Universal Robots PolyScope program: DAS428_958_02_MAR_21_DAS_lado_derecho_jig2.urp

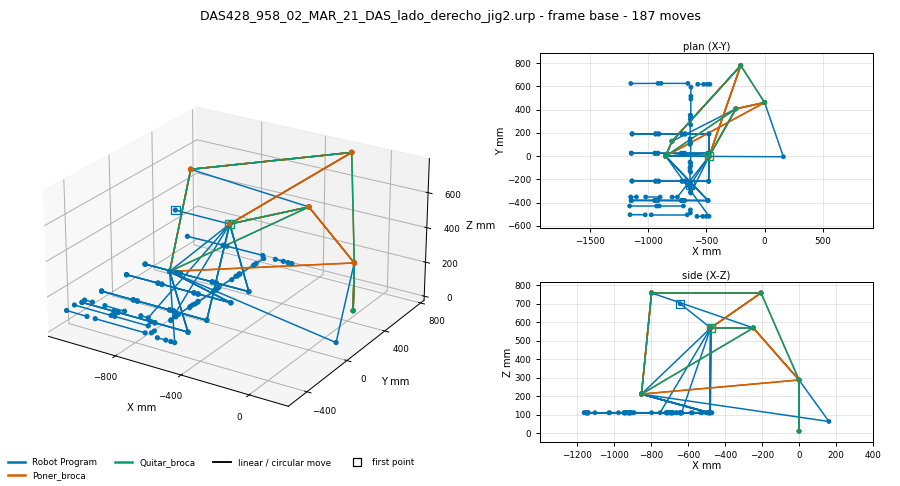
[picture p0: tool path of DAS428_958_02_MAR_21_DAS_lado_derecho_jig2.urp in frame base, 187 of 372 moves have a stored position in this frame; points joined in program order, loops and branches not executed]
Program DAS428_958_02_MAR_21_DAS_lado_derecho_jig2 (installation=instalacion_26_FEB_21 directory=/programs/jig2/derecha createdIn=5.6.0.90886 lastSavedIn=5.6.0.90886 robotSerialNumber=20195001785)
Calibrated DH parameters: a=[0.000107, -0.568984, -0.552934, -0.00001, -0.000063, 0]; d=[0.180718, -257.998067, 200.685024, 57.48776, 0.119923, 0.115353]; alpha=[1.571119, 0.000876, -0.002498, 1.571178, -1.570523, 0]; deltaTheta=[0, -0.378191, 0.631587, -0.253396, 0, 0]
Robot Program (runOnlyOnce=false)
  Folder Variables
    bajada_broca := p[0,0,-0.008,0,0,0]
    barrenos_menos1 := 0
    barreno_actual := 0
    posicion := p[0,0,300,0,0,0]
    cambiar_broca := False
    barrenos_hechos := 0
    eje7 := 0
    Wait Sleep waitTime=0.5
  Folder Home
    Wait Sleep waitTime=0.3
    MoveL speed 250 mm/s, acceleration 1200 mm/s^2 (useActiveTCP=true) feature=Base
      Waypoint Traslacion: TCP in base x=-641.047 y=-250.866 z=699.551 mm, rx=2.5572 ry=-1.7056 rz=-0.147 rad; joints [-0.465, -94.502, 70.676, 17.843, -302.102, -0.163] deg; TCP offset x=0.411 y=-218.298 z=37.994 mm, rx=1.558 ry=-0.1255 rz=0.1212 rad
      Waypoint Home2: TCP in base x=-476.229 y=0 z=568.737 mm, rx=2.0263 ry=-2.3929 rz=-0.0208 rad; joints [-32.551, -116.469, 98.413, 17.843, -302.102, -0.163] deg; TCP offset x=0.411 y=-218.298 z=37.994 mm, rx=1.558 ry=-0.1255 rz=0.1212 rad
      Waypoint Home3: TCP in base x=-850.182 y=0 z=211.32 mm, rx=-2.0297 ry=2.3968 rz=0.0066 rad; joints [-14.374, -75.698, 98.757, -22.649, -284.037, -0.192] deg; TCP offset x=0.411 y=-218.298 z=37.994 mm, rx=1.558 ry=-0.1255 rz=0.1212 rad
      Waypoint Home4: TCP in base x=-850.182 y=0 z=211.32 mm, rx=-2.0297 ry=2.3968 rz=0.0066 rad; joints [-14.374, -75.698, 98.757, -22.649, -284.037, -0.192] deg; TCP offset x=0.411 y=-218.298 z=37.994 mm, rx=1.558 ry=-0.1255 rz=0.1212 rad
      Waypoint PosicionApagado: TCP in base x=162.343 y=-4.969 z=63.23 mm, rx=-1.8392 ry=0.2253 rz=0.1717 rad; joints [89.997, -89.982, 149.522, 14.976, -265, 0.001] deg
      Waypoint Precambio_broca: TCP in base x=0.83 y=461.518 z=287.521 mm, rx=-0.2218 ry=-3.132 rz=0.0004 rad; joints [-125.124, -120.118, 128.54, -7.699, -306.118, -0.232] deg; TCP offset x=0.411 y=-218.298 z=37.994 mm, rx=1.558 ry=-0.1255 rz=0.1212 rad
      Waypoint yendo1: TCP in base x=-246.137 y=407.69 z=568.737 mm, rx=-0.5894 ry=3.0844 rz=0.0228 rad; joints [-91.431, -116.469, 98.413, 17.843, -302.102, -0.163] deg
      Waypoint Precam_bro1: TCP in base x=-795.771 y=128.511 z=757.632 mm, rx=1.5534 ry=-2.1987 rz=-0.8089 rad; joints [-24.356, -99.239, 84.164, -22.649, -284.037, -0.192] deg; TCP offset x=0.411 y=-218.298 z=37.994 mm, rx=1.558 ry=-0.1255 rz=0.1212 rad
      Waypoint Precam_bro2: TCP in base x=-204.472 y=779.716 z=757.632 mm, rx=-0.1114 ry=2.934 rz=1.0184 rad; joints [-90.488, -99.239, 84.164, -22.649, -284.037, -0.192] deg
    SafeHome (positionOptionType=SPEED_AND_ACCELERATION speed=1.047198 acceleration=1.396263 nextMotionTime=2)
    SuppressedNode
      If eje7≟3
        MoveL speed 250 mm/s, acceleration 1200 mm/s^2 (useActiveTCP=true) feature=Base
          MoveDirectionNode (selectedDirection=ZPlus)
            Until DISTANCE (allowActions=false deceleration=3 distanceNodeType=STOP) Distance=0.1; motionParameters(blendRadius=0)
          Waypoint Home3: TCP in base x=-850.182 y=0 z=211.32 mm, rx=-2.0297 ry=2.3968 rz=0.0066 rad; joints [-14.374, -75.698, 98.757, -22.649, -284.037, -0.192] deg
    SuppressedNode
      MoveL speed 250 mm/s, acceleration 1200 mm/s^2 (useActiveTCP=true) feature=Base
        Waypoint home_trans: TCP in base x=-171.077 y=546.65 z=109.574 mm, rx=0.1544 ry=3.1247 rz=-0.2011 rad; joints [-91.802, -93.053, 127.954, -27.005, -275.278, -0.192] deg; TCP offset x=0.411 y=-218.298 z=37.994 mm, rx=1.558 ry=-0.1255 rz=0.1212 rad
    Wait Sleep waitTime=0.3
    iniciando_prog := True
    Call Poner_broca
  Folder Posicion2
    Folder Inicio
      eje7 := 2
      MoveL speed 250 mm/s, acceleration 1200 mm/s^2 (useActiveTCP=true) feature=Base
        Waypoint Home2: TCP in base x=-476.229 y=0 z=568.737 mm, rx=2.0263 ry=-2.3929 rz=-0.0208 rad; joints [-32.551, -116.469, 98.413, 17.843, -302.102, -0.163] deg
    Folder SeatTracks
      Folder Broca_1
        Folder Linea1
          Folder Marcar_puntos
            MoveL speed 100 mm/s, acceleration 500 mm/s^2 (useActiveTCP=true) feature=Base
              Waypoint Home2: TCP in base x=-476.229 y=0 z=568.737 mm, rx=2.0263 ry=-2.3929 rz=-0.0208 rad; joints [-32.551, -116.469, 98.413, 17.843, -302.102, -0.163] deg
              SuppressedNode
                Folder var
                  barrenos_hechos := 10
                  eje7 := 2
                  cambiar_broca := False
                  iniciando_prog := False
              SuppressedNode
                iniciando_prog := False
              SuppressedNode
                Call Poner_broca
              Waypoint Linea1_A: TCP in base x=-480.065 y=-215.567 z=110.155 mm, rx=2.0263 ry=-2.3929 rz=-0.0208 rad; joints [7.208, -100.641, 136.552, -36.178, -262.472, -0.269] deg; TCP offset x=0.411 y=-218.298 z=37.994 mm, rx=1.558 ry=-0.1255 rz=0.1212 rad
              Waypoint Linea1_B: TCP in base x=-683.26 y=-215.006 z=110.473 mm, rx=2.0263 ry=-2.3929 rz=-0.0208 rad; joints [4.504, -82.11, 118.563, -36.711, -265.183, -0.242] deg
              Waypoint Linea1_C: TCP in base x=-708.66 y=-214.986 z=110.511 mm, rx=2.0264 ry=-2.3929 rz=-0.0208 rad; joints [4.302, -80.013, 116.028, -36.271, -265.387, -0.241] deg
              Waypoint Linea1_D: TCP in base x=-911.542 y=-214.533 z=110.306 mm, rx=2.0263 ry=-2.3929 rz=-0.0209 rad; joints [3.146, -63.772, 93.392, -29.877, -266.531, -0.235] deg
              Waypoint Linea1_E: TCP in base x=-936.518 y=-214.589 z=110.515 mm, rx=2.0263 ry=-2.3929 rz=-0.0209 rad; joints [3.051, -61.764, 90.233, -28.728, -266.622, -0.234] deg
              Waypoint Linea1_F: TCP in base x=-1139.514 y=-213.881 z=110.127 mm, rx=2.0263 ry=-2.3929 rz=-0.0209 rad; joints [2.389, -43.641, 59.472, -16.09, -267.256, -0.236] deg
          Folder AB
            'desbaste_inicial'
            bajada_broca := p[0,0,-0.008,0,0,0]
            barrenos_menos1 := 8
            barreno_actual := 0
            Loop While (checkContinuously=false) expression=barreno_actual≤barrenos_menos1
              Folder Perforacion
                MoveL speed 100 mm/s, acceleration 500 mm/s^2 (useActiveTCP=true) feature=Base
                  internos := interpolate_pose(Linea1_A, Linea1_B, barreno_actual/barrenos_menos1)
                  Waypoint Waypoint (Variable): variable=internos
                  'desbaste_inicial'
                  bajada_broca := p[0,0,-0.008,0,0,0]
                  bajada := p[0,0,0.008,0,0,0]
                  MoveDirectionNode (selectedDirection=ZMinus toolParams=0.03, 0.035)
                    Until DISTANCE (allowActions=false deceleration=3 distanceNodeType=STOP) Distance=0.076; motionParameters(blendRadius=0)
                  Popup Message (haltProgram=false message=punto contacto alanzdo inputType=Text)
                  MoveDirectionNode (selectedDirection=ZPlus toolParams=0.003, 0.005)
                    Until DISTANCE (allowActions=false deceleration=3 distanceNodeType=STOP) Distance=0.002; motionParameters(blendRadius=0)
                  Wait Sleep waitTime=0.3
                  Set DigitalOutput pin=config_out[1]; digitalValue=1
                  Wait Sleep waitTime=0.3
                  Loop Counting (count=3) loopVariable(name=Loop_39)
                    bajar := pose_add(get_actual_tcp_pose(), bajada_broca)
                    Waypoint Waypoint (Variable): motionParameters(jointSpeed=1.047198 jointAcceleration=1.396263 cartesianSpeed=0.001 cartesianAcceleration=0.005); variable=bajar
                    subir := pose_sub(get_actual_tcp_pose(), bajada_broca)
                    Waypoint Waypoint (Variable): motionParameters(jointSpeed=1.047198 jointAcceleration=1.396263 cartesianSpeed=0.005 cartesianAcceleration=0.01); variable=subir
                    bajada_broca := pose_sub(bajada_broca, bajada)
                  MoveDirectionNode (selectedDirection=ZPlus toolParams=0.03, 0.035)
                    Until DISTANCE (allowActions=false deceleration=3 distanceNodeType=STOP) Distance=0.06; motionParameters(blendRadius=0)
                  Set DigitalOutput pin=config_out[1]; digitalValue=0
                  barreno_actual := barreno_actual+1
                  Call Quitar_broca
                  Call Poner_broca
          Folder CD
            'desbaste_inicial'
            bajada_broca := p[0,0,-0.008,0,0,0]
            barrenos_menos1 := 8
            barreno_actual := 0
            Loop While (checkContinuously=false) expression=barreno_actual≤barrenos_menos1
              Folder Perforacion
                MoveL speed 100 mm/s, acceleration 500 mm/s^2 (useActiveTCP=true) feature=Base
                  internos := interpolate_pose(Linea1_C, Linea1_D, barreno_actual/barrenos_menos1)
                  Waypoint Waypoint (Variable): variable=internos
                  'desbaste_inicial'
                  bajada_broca := p[0,0,-0.008,0,0,0]
                  bajada := p[0,0,0.008,0,0,0]
                  MoveDirectionNode (selectedDirection=ZMinus toolParams=0.03, 0.035)
                    Until DISTANCE (allowActions=false deceleration=3 distanceNodeType=STOP) Distance=0.076; motionParameters(blendRadius=0)
                  Popup Message (haltProgram=false message=punto contacto alanzdo inputType=Text)
                  MoveDirectionNode (selectedDirection=ZPlus toolParams=0.003, 0.005)
                    Until DISTANCE (allowActions=false deceleration=3 distanceNodeType=STOP) Distance=0.002; motionParameters(blendRadius=0)
                  Wait Sleep waitTime=0.3
                  Set DigitalOutput pin=config_out[1]; digitalValue=1
                  Wait Sleep waitTime=0.3
                  Loop Counting (count=3) loopVariable(name=Loop_56)
                    bajar := pose_add(get_actual_tcp_pose(), bajada_broca)
                    Waypoint Waypoint (Variable): motionParameters(jointSpeed=1.047198 jointAcceleration=1.396263 cartesianSpeed=0.001 cartesianAcceleration=0.005); variable=bajar
                    subir := pose_sub(get_actual_tcp_pose(), bajada_broca)
                    Waypoint Waypoint (Variable): motionParameters(jointSpeed=1.047198 jointAcceleration=1.396263 cartesianSpeed=0.005 cartesianAcceleration=0.01); variable=subir
                    bajada_broca := pose_sub(bajada_broca, bajada)
                  MoveDirectionNode (selectedDirection=ZPlus toolParams=0.03, 0.035)
                    Until DISTANCE (allowActions=false deceleration=3 distanceNodeType=STOP) Distance=0.06; motionParameters(blendRadius=0)
                  Set DigitalOutput pin=config_out[1]; digitalValue=0
                  barreno_actual := barreno_actual+1
                  Call Quitar_broca
                  Call Poner_broca
          Folder EF
            'desbaste_inicial'
            bajada_broca := p[0,0,-0.008,0,0,0]
            barrenos_menos1 := 8
            barreno_actual := 0
            Loop While (checkContinuously=false) expression=barreno_actual≤barrenos_menos1
              Folder Perforacion
                MoveL speed 100 mm/s, acceleration 500 mm/s^2 (useActiveTCP=true) feature=Base
                  internos := interpolate_pose(Linea1_E, Linea1_F, barreno_actual/barrenos_menos1)
                  Waypoint Waypoint (Variable): variable=internos
                  'desbaste_inicial'
                  bajada_broca := p[0,0,-0.008,0,0,0]
                  bajada := p[0,0,0.008,0,0,0]
                  MoveDirectionNode (selectedDirection=ZMinus toolParams=0.03, 0.035)
                    Until DISTANCE (allowActions=false deceleration=3 distanceNodeType=STOP) Distance=0.067; motionParameters(blendRadius=0)
                  Popup Message (haltProgram=false message=punto contacto alanzdo inputType=Text)
                  MoveDirectionNode (selectedDirection=ZPlus toolParams=0.003, 0.005)
                    Until DISTANCE (allowActions=false deceleration=3 distanceNodeType=STOP) Distance=0.002; motionParameters(blendRadius=0)
                  Wait Sleep waitTime=0.3
                  Set DigitalOutput pin=config_out[1]; digitalValue=1
                  Wait Sleep waitTime=0.3
                  Loop Counting (count=3) loopVariable(name=Loop_61)
                    bajar := pose_add(get_actual_tcp_pose(), bajada_broca)
                    Waypoint Waypoint (Variable): motionParameters(jointSpeed=1.047198 jointAcceleration=1.396263 cartesianSpeed=0.001 cartesianAcceleration=0.005); variable=bajar
                    subir := pose_sub(get_actual_tcp_pose(), bajada_broca)
                    Waypoint Waypoint (Variable): motionParameters(jointSpeed=1.047198 jointAcceleration=1.396263 cartesianSpeed=0.005 cartesianAcceleration=0.01); variable=subir
                    bajada_broca := pose_sub(bajada_broca, bajada)
                  MoveDirectionNode (selectedDirection=ZPlus toolParams=0.03, 0.035)
                    Until DISTANCE (allowActions=false deceleration=3 distanceNodeType=STOP) Distance=0.06; motionParameters(blendRadius=0)
                  Set DigitalOutput pin=config_out[1]; digitalValue=0
                  barreno_actual := barreno_actual+1
                  Call Quitar_broca
                  Call Poner_broca
        Popup Message (haltProgram=false message=Linea1 con chica Terminada! inputType=Text)
        Folder Linea2
          Folder Marcar_puntos
            MoveL speed 100 mm/s, acceleration 500 mm/s^2 (useActiveTCP=true) feature=Base
              Waypoint Home2: TCP in base x=-476.229 y=0 z=568.737 mm, rx=2.0263 ry=-2.3929 rz=-0.0208 rad; joints [-32.551, -116.469, 98.413, 17.843, -302.102, -0.163] deg; TCP offset x=0.411 y=-218.298 z=37.994 mm, rx=1.558 ry=-0.1255 rz=0.1212 rad
              Waypoint Linea2_A: TCP in base x=-478.57 y=191.006 z=110.523 mm, rx=2.0263 ry=-2.3928 rz=-0.0209 rad; joints [-57.982, -102.694, 138.014, -35.673, -327.66, 0.098] deg; TCP offset x=0.411 y=-218.298 z=37.994 mm, rx=1.558 ry=-0.1255 rz=0.1212 rad
              Waypoint Linea2_B: TCP in base x=-681.936 y=191.002 z=110.452 mm, rx=2.0263 ry=-2.3929 rz=-0.0209 rad; joints [-37.869, -83.103, 119.731, -36.904, -307.554, -0.038] deg
              Waypoint Linea2_C: TCP in base x=-707.214 y=190.995 z=110.603 mm, rx=2.0262 ry=-2.3929 rz=-0.0208 rad; joints [-36.266, -80.967, 117.182, -36.489, -305.951, -0.043] deg
              Waypoint Linea2_D: TCP in base x=-910.192 y=191.479 z=110.348 mm, rx=2.0262 ry=-2.3928 rz=-0.0209 rad; joints [-27.02, -64.45, 94.432, -30.243, -296.696, -0.089] deg
              Waypoint Linea2_E: TCP in base x=-935.62 y=191.519 z=110.454 mm, rx=2.0261 ry=-2.3928 rz=-0.021 rad; joints [-26.177, -62.39, 91.226, -29.103, -295.849, -0.094] deg
              Waypoint Linea2_F: TCP in base x=-1138.395 y=191.499 z=110.212 mm, rx=2.0262 ry=-2.3928 rz=-0.021 rad; joints [-20.933, -44.304, 60.66, -16.618, -290.578, -0.121] deg
          Folder AB
            'desbaste_inicial'
            bajada_broca := p[0,0,-0.008,0,0,0]
            barrenos_menos1 := 8
            barreno_actual := 0
            Loop While (checkContinuously=false) expression=barreno_actual≤barrenos_menos1
              Folder Perforacion
                MoveL speed 100 mm/s, acceleration 500 mm/s^2 (useActiveTCP=true) feature=Base
                  internos := interpolate_pose(Linea2_A, Linea2_B, barreno_actual/barrenos_menos1)
                  Waypoint Waypoint (Variable): variable=internos
                  'desbaste_inicial'
                  bajada_broca := p[0,0,-0.008,0,0,0]
                  bajada := p[0,0,0.008,0,0,0]
                  MoveDirectionNode (selectedDirection=ZMinus toolParams=0.03, 0.035)
                    Until DISTANCE (allowActions=false deceleration=3 distanceNodeType=STOP) Distance=0.076; motionParameters(blendRadius=0)
                  Popup Message (haltProgram=false message=punto contacto alanzdo inputType=Text)
                  MoveDirectionNode (selectedDirection=ZPlus toolParams=0.003, 0.005)
                    Until DISTANCE (allowActions=false deceleration=3 distanceNodeType=STOP) Distance=0.002; motionParameters(blendRadius=0)
                  Wait Sleep waitTime=0.3
                  Set DigitalOutput pin=config_out[1]; digitalValue=1
                  Wait Sleep waitTime=0.3
                  Loop Counting (count=3) loopVariable(name=Loop_63)
                    bajar := pose_add(get_actual_tcp_pose(), bajada_broca)
                    Waypoint Waypoint (Variable): motionParameters(jointSpeed=1.047198 jointAcceleration=1.396263 cartesianSpeed=0.001 cartesianAcceleration=0.005); variable=bajar
                    subir := pose_sub(get_actual_tcp_pose(), bajada_broca)
                    Waypoint Waypoint (Variable): motionParameters(jointSpeed=1.047198 jointAcceleration=1.396263 cartesianSpeed=0.005 cartesianAcceleration=0.01); variable=subir
                    bajada_broca := pose_sub(bajada_broca, bajada)
                  MoveDirectionNode (selectedDirection=ZPlus toolParams=0.03, 0.035)
                    Until DISTANCE (allowActions=false deceleration=3 distanceNodeType=STOP) Distance=0.06; motionParameters(blendRadius=0)
                  Set DigitalOutput pin=config_out[1]; digitalValue=0
                  barreno_actual := barreno_actual+1
                  Call Quitar_broca
                  Call Poner_broca
          Folder CD
            'desbaste_inicial'
            bajada_broca := p[0,0,-0.008,0,0,0]
            barrenos_menos1 := 8
            barreno_actual := 0
            Loop While (checkContinuously=false) expression=barreno_actual≤barrenos_menos1
              Folder Perforacion
                MoveL speed 100 mm/s, acceleration 500 mm/s^2 (useActiveTCP=true) feature=Base
                  internos := interpolate_pose(Linea2_C, Linea2_D, barreno_actual/barrenos_menos1)
                  Waypoint Waypoint (Variable): variable=internos
                  'desbaste_inicial'
                  bajada_broca := p[0,0,-0.008,0,0,0]
                  bajada := p[0,0,0.008,0,0,0]
                  MoveDirectionNode (selectedDirection=ZMinus toolParams=0.03, 0.035)
                    Until DISTANCE (allowActions=false deceleration=3 distanceNodeType=STOP) Distance=0.076; motionParameters(blendRadius=0)
                  Popup Message (haltProgram=false message=punto contacto alanzdo inputType=Text)
                  MoveDirectionNode (selectedDirection=ZPlus toolParams=0.003, 0.005)
                    Until DISTANCE (allowActions=false deceleration=3 distanceNodeType=STOP) Distance=0.002; motionParameters(blendRadius=0)
                  Wait Sleep waitTime=0.3
                  Set DigitalOutput pin=config_out[1]; digitalValue=1
                  Wait Sleep waitTime=0.3
                  Loop Counting (count=3) loopVariable(name=Loop_65)
                    bajar := pose_add(get_actual_tcp_pose(), bajada_broca)
                    Waypoint Waypoint (Variable): motionParameters(jointSpeed=1.047198 jointAcceleration=1.396263 cartesianSpeed=0.001 cartesianAcceleration=0.005); variable=bajar
                    subir := pose_sub(get_actual_tcp_pose(), bajada_broca)
                    Waypoint Waypoint (Variable): motionParameters(jointSpeed=1.047198 jointAcceleration=1.396263 cartesianSpeed=0.005 cartesianAcceleration=0.01); variable=subir
                    bajada_broca := pose_sub(bajada_broca, bajada)
                  MoveDirectionNode (selectedDirection=ZPlus toolParams=0.03, 0.035)
                    Until DISTANCE (allowActions=false deceleration=3 distanceNodeType=STOP) Distance=0.06; motionParameters(blendRadius=0)
                  Set DigitalOutput pin=config_out[1]; digitalValue=0
                  barreno_actual := barreno_actual+1
                  Call Quitar_broca
                  Call Poner_broca
          Folder EF
            'desbaste_inicial'
            bajada_broca := p[0,0,-0.008,0,0,0]
            barrenos_menos1 := 8
            barreno_actual := 0
            Loop While (checkContinuously=false) expression=barreno_actual≤barrenos_menos1
              Folder Perforacion
                MoveL speed 100 mm/s, acceleration 500 mm/s^2 (useActiveTCP=true) feature=Base
                  internos := interpolate_pose(Linea2_E, Linea2_F, barreno_actual/barrenos_menos1)
                  Waypoint Waypoint (Variable): variable=internos
                  'desbaste_inicial'
                  bajada_broca := p[0,0,-0.008,0,0,0]
                  bajada := p[0,0,0.008,0,0,0]
                  MoveDirectionNode (selectedDirection=ZMinus toolParams=0.03, 0.035)
                    Until DISTANCE (allowActions=false deceleration=3 distanceNodeType=STOP) Distance=0.076; motionParameters(blendRadius=0)
                  Popup Message (haltProgram=false message=punto contacto alanzdo inputType=Text)
                  MoveDirectionNode (selectedDirection=ZPlus toolParams=0.003, 0.005)
                    Until DISTANCE (allowActions=false deceleration=3 distanceNodeType=STOP) Distance=0.002; motionParameters(blendRadius=0)
                  Wait Sleep waitTime=0.3
                  Set DigitalOutput pin=config_out[1]; digitalValue=1
                  Wait Sleep waitTime=0.3
                  Loop Counting (count=3) loopVariable(name=Loop_67)
                    bajar := pose_add(get_actual_tcp_pose(), bajada_broca)
                    Waypoint Waypoint (Variable): motionParameters(jointSpeed=1.047198 jointAcceleration=1.396263 cartesianSpeed=0.001 cartesianAcceleration=0.005); variable=bajar
                    subir := pose_sub(get_actual_tcp_pose(), bajada_broca)
                    Waypoint Waypoint (Variable): motionParameters(jointSpeed=1.047198 jointAcceleration=1.396263 cartesianSpeed=0.005 cartesianAcceleration=0.01); variable=subir
                    bajada_broca := pose_sub(bajada_broca, bajada)
                  MoveDirectionNode (selectedDirection=ZPlus toolParams=0.03, 0.035)
                    Until DISTANCE (allowActions=false deceleration=3 distanceNodeType=STOP) Distance=0.06; motionParameters(blendRadius=0)
                  Set DigitalOutput pin=config_out[1]; digitalValue=0
                  barreno_actual := barreno_actual+1
                  If barreno_actual>barrenos_menos1
                    cambiar_broca := True
                  Call Quitar_broca
                  Call Poner_broca
        Popup Message (haltProgram=false message=Linea2 con chica Terminada! inputType=Text)
      Folder Broca_2
        Folder Linea1
          Folder Marcar_puntos
            MoveL speed 100 mm/s, acceleration 500 mm/s^2 (useActiveTCP=true) feature=Base
              Waypoint Home2: TCP in base x=-476.229 y=0 z=568.737 mm, rx=2.0263 ry=-2.3929 rz=-0.0208 rad; joints [-32.551, -116.469, 98.413, 17.843, -302.102, -0.163] deg; TCP offset x=0.411 y=-218.298 z=37.994 mm, rx=1.558 ry=-0.1255 rz=0.1212 rad
              SuppressedNode
                Folder var
                  barrenos_hechos := 10
                  eje7 := 2
                  cambiar_broca := False
                  iniciando_prog := False
              SuppressedNode
                iniciando_prog := True
              SuppressedNode
                Call Poner_broca
              Waypoint Linea1_A: TCP in base x=-480.065 y=-215.567 z=110.155 mm, rx=2.0263 ry=-2.3929 rz=-0.0208 rad; joints [7.208, -100.641, 136.552, -36.178, -262.472, -0.269] deg; TCP offset x=0.411 y=-218.298 z=37.994 mm, rx=1.558 ry=-0.1255 rz=0.1212 rad
              Waypoint Linea1_B: TCP in base x=-683.26 y=-215.006 z=110.473 mm, rx=2.0263 ry=-2.3929 rz=-0.0208 rad; joints [4.504, -82.11, 118.563, -36.711, -265.183, -0.242] deg
              Waypoint Linea1_C: TCP in base x=-708.66 y=-214.986 z=110.511 mm, rx=2.0264 ry=-2.3929 rz=-0.0208 rad; joints [4.302, -80.013, 116.028, -36.271, -265.387, -0.241] deg
              Waypoint Linea1_D: TCP in base x=-911.542 y=-214.533 z=110.306 mm, rx=2.0263 ry=-2.3929 rz=-0.0209 rad; joints [3.146, -63.772, 93.392, -29.877, -266.531, -0.235] deg
              Waypoint Linea1_E: TCP in base x=-936.518 y=-214.589 z=110.515 mm, rx=2.0263 ry=-2.3929 rz=-0.0209 rad; joints [3.051, -61.764, 90.233, -28.728, -266.622, -0.234] deg
              Waypoint Linea1_F: TCP in base x=-1139.514 y=-213.881 z=110.127 mm, rx=2.0263 ry=-2.3929 rz=-0.0209 rad; joints [2.389, -43.641, 59.472, -16.09, -267.256, -0.236] deg
          Folder AB
            'desbaste_inicial'
            bajada_broca := p[0,0,-0.012,0,0,0]
            barrenos_menos1 := 8
            barreno_actual := 0
            Loop While (checkContinuously=false) expression=barreno_actual≤barrenos_menos1
              Folder Perforacion
                MoveL speed 100 mm/s, acceleration 500 mm/s^2 (useActiveTCP=true) feature=Base
                  internos := interpolate_pose(Linea1_A, Linea1_B, barreno_actual/barrenos_menos1)
                  Waypoint Waypoint (Variable): variable=internos
                  'desbaste_inicial'
                  bajada_broca := p[0,0,-0.012,0,0,0]
                  bajada := p[0,0,0.012,0,0,0]
                  MoveDirectionNode (selectedDirection=ZMinus toolParams=0.03, 0.035)
                    Until DISTANCE (allowActions=false deceleration=3 distanceNodeType=STOP) Distance=0.072; motionParameters(blendRadius=0)
                  Popup Message (haltProgram=false message=punto contacto alanzdo inputType=Text)
                  MoveDirectionNode (selectedDirection=ZPlus toolParams=0.003, 0.005)
                    Until DISTANCE (allowActions=false deceleration=3 distanceNodeType=STOP) Distance=0.002; motionParameters(blendRadius=0)
                  Wait Sleep waitTime=0.3
                  Set DigitalOutput pin=config_out[1]; digitalValue=1
                  Wait Sleep waitTime=0.3
                  Loop Counting (count=2) loopVariable(name=Loop_69)
                    bajar := pose_add(get_actual_tcp_pose(), bajada_broca)
                    Waypoint Waypoint (Variable): motionParameters(jointSpeed=1.047198 jointAcceleration=1.396263 cartesianSpeed=0.001 cartesianAcceleration=0.005); variable=bajar
                    subir := pose_sub(get_actual_tcp_pose(), bajada_broca)
                    Waypoint Waypoint (Variable): motionParameters(jointSpeed=1.047198 jointAcceleration=1.396263 cartesianSpeed=0.005 cartesianAcceleration=0.01); variable=subir
                    bajada_broca := pose_sub(bajada_broca, bajada)
                  MoveDirectionNode (selectedDirection=ZPlus toolParams=0.03, 0.035)
                    Until DISTANCE (allowActions=false deceleration=3 distanceNodeType=STOP) Distance=0.06; motionParameters(blendRadius=0)
                  Set DigitalOutput pin=config_out[1]; digitalValue=0
                  barreno_actual := barreno_actual+1
                  Call Quitar_broca
                  Call Poner_broca
          Folder CD
            'desbaste_inicial'
            bajada_broca := p[0,0,-0.012,0,0,0]
            barrenos_menos1 := 8
            barreno_actual := 0
            Loop While (checkContinuously=false) expression=barreno_actual≤barrenos_menos1
              Folder Perforacion
                MoveL speed 100 mm/s, acceleration 500 mm/s^2 (useActiveTCP=true) feature=Base
                  internos := interpolate_pose(Linea1_C, Linea1_D, barreno_actual/barrenos_menos1)
                  Waypoint Waypoint (Variable): variable=internos
                  'desbaste_inicial'
                  bajada_broca := p[0,0,-0.012,0,0,0]
                  bajada := p[0,0,0.012,0,0,0]
                  MoveDirectionNode (selectedDirection=ZMinus toolParams=0.03, 0.035)
                    Until DISTANCE (allowActions=false deceleration=3 distanceNodeType=STOP) Distance=0.072; motionParameters(blendRadius=0)
                  Popup Message (haltProgram=false message=punto contacto alanzdo inputType=Text)
                  MoveDirectionNode (selectedDirection=ZPlus toolParams=0.003, 0.005)
                    Until DISTANCE (allowActions=false deceleration=3 distanceNodeType=STOP) Distance=0.002; motionParameters(blendRadius=0)
                  Wait Sleep waitTime=0.3
                  Set DigitalOutput pin=config_out[1]; digitalValue=1
                  Wait Sleep waitTime=0.3
                  Loop Counting (count=2) loopVariable(name=Loop_71)
                    bajar := pose_add(get_actual_tcp_pose(), bajada_broca)
                    Waypoint Waypoint (Variable): motionParameters(jointSpeed=1.047198 jointAcceleration=1.396263 cartesianSpeed=0.001 cartesianAcceleration=0.005); variable=bajar
                    subir := pose_sub(get_actual_tcp_pose(), bajada_broca)
                    Waypoint Waypoint (Variable): motionParameters(jointSpeed=1.047198 jointAcceleration=1.396263 cartesianSpeed=0.005 cartesianAcceleration=0.01); variable=subir
                    bajada_broca := pose_sub(bajada_broca, bajada)
                  MoveDirectionNode (selectedDirection=ZPlus toolParams=0.03, 0.035)
                    Until DISTANCE (allowActions=false deceleration=3 distanceNodeType=STOP) Distance=0.06; motionParameters(blendRadius=0)
                  Set DigitalOutput pin=config_out[1]; digitalValue=0
                  barreno_actual := barreno_actual+1
                  Call Quitar_broca
                  Call Poner_broca
          Folder EF
            'desbaste_inicial'
            bajada_broca := p[0,0,-0.012,0,0,0]
            barrenos_menos1 := 8
            barreno_actual := 0
            Loop While (checkContinuously=false) expression=barreno_actual≤barrenos_menos1
              Folder Perforacion
                MoveL speed 100 mm/s, acceleration 500 mm/s^2 (useActiveTCP=true) feature=Base
                  internos := interpolate_pose(Linea1_E, Linea1_F, barreno_actual/barrenos_menos1)
                  Waypoint Waypoint (Variable): variable=internos
                  'desbaste_inicial'
                  bajada_broca := p[0,0,-0.012,0,0,0]
                  bajada := p[0,0,0.012,0,0,0]
                  MoveDirectionNode (selectedDirection=ZMinus toolParams=0.03, 0.035)
                    Until DISTANCE (allowActions=false deceleration=3 distanceNodeType=STOP) Distance=0.072; motionParameters(blendRadius=0)
                  Popup Message (haltProgram=false message=punto contacto alanzdo inputType=Text)
                  MoveDirectionNode (selectedDirection=ZPlus toolParams=0.003, 0.005)
                    Until DISTANCE (allowActions=false deceleration=3 distanceNodeType=STOP) Distance=0.002; motionParameters(blendRadius=0)
                  Wait Sleep waitTime=0.3
                  Set DigitalOutput pin=config_out[1]; digitalValue=1
                  Wait Sleep waitTime=0.3
                  Loop Counting (count=2) loopVariable(name=Loop_73)
                    bajar := pose_add(get_actual_tcp_pose(), bajada_broca)
                    Waypoint Waypoint (Variable): motionParameters(jointSpeed=1.047198 jointAcceleration=1.396263 cartesianSpeed=0.001 cartesianAcceleration=0.005); variable=bajar
                    subir := pose_sub(get_actual_tcp_pose(), bajada_broca)
                    Waypoint Waypoint (Variable): motionParameters(jointSpeed=1.047198 jointAcceleration=1.396263 cartesianSpeed=0.005 cartesianAcceleration=0.01); variable=subir
                    bajada_broca := pose_sub(bajada_broca, bajada)
                  MoveDirectionNode (selectedDirection=ZPlus toolParams=0.03, 0.035)
                    Until DISTANCE (allowActions=false deceleration=3 distanceNodeType=STOP) Distance=0.06; motionParameters(blendRadius=0)
                  Set DigitalOutput pin=config_out[1]; digitalValue=0
                  barreno_actual := barreno_actual+1
                  Call Quitar_broca
                  Call Poner_broca
        Popup Message (haltProgram=false message=Linea1 con media Terminada! inputType=Text)
        Folder Linea2
          Folder Marcar_puntos
            MoveL speed 100 mm/s, acceleration 500 mm/s^2 (useActiveTCP=true) feature=Base
              Waypoint Home2: TCP in base x=-476.229 y=0 z=568.737 mm, rx=2.0263 ry=-2.3929 rz=-0.0208 rad; joints [-32.551, -116.469, 98.413, 17.843, -302.102, -0.163] deg; TCP offset x=0.411 y=-218.298 z=37.994 mm, rx=1.558 ry=-0.1255 rz=0.1212 rad
              Waypoint Linea2_A: TCP in base x=-478.57 y=191.006 z=110.523 mm, rx=2.0263 ry=-2.3928 rz=-0.0209 rad; joints [-57.982, -102.694, 138.014, -35.673, -327.66, 0.098] deg; TCP offset x=0.411 y=-218.298 z=37.994 mm, rx=1.558 ry=-0.1255 rz=0.1212 rad
              Waypoint Linea2_B: TCP in base x=-681.936 y=191.002 z=110.452 mm, rx=2.0263 ry=-2.3929 rz=-0.0209 rad; joints [-37.869, -83.103, 119.731, -36.904, -307.554, -0.038] deg
              Waypoint Linea2_C: TCP in base x=-707.214 y=190.995 z=110.603 mm, rx=2.0262 ry=-2.3929 rz=-0.0208 rad; joints [-36.266, -80.967, 117.182, -36.489, -305.951, -0.043] deg
              Waypoint Linea2_D: TCP in base x=-910.192 y=191.479 z=110.348 mm, rx=2.0262 ry=-2.3928 rz=-0.0209 rad; joints [-27.02, -64.45, 94.432, -30.243, -296.696, -0.089] deg
              Waypoint Linea2_E: TCP in base x=-935.62 y=191.519 z=110.454 mm, rx=2.0261 ry=-2.3928 rz=-0.021 rad; joints [-26.177, -62.39, 91.226, -29.103, -295.849, -0.094] deg
              Waypoint Linea2_F: TCP in base x=-1138.395 y=191.499 z=110.212 mm, rx=2.0262 ry=-2.3928 rz=-0.021 rad; joints [-20.933, -44.304, 60.66, -16.618, -290.578, -0.121] deg
          Folder AB
            'desbaste_inicial'
            bajada_broca := p[0,0,-0.012,0,0,0]
            barrenos_menos1 := 8
            barreno_actual := 0
            Loop While (checkContinuously=false) expression=barreno_actual≤barrenos_menos1
              Folder Perforacion
                MoveL speed 100 mm/s, acceleration 500 mm/s^2 (useActiveTCP=true) feature=Base
                  internos := interpolate_pose(Linea2_A, Linea2_B, barreno_actual/barrenos_menos1)
                  Waypoint Waypoint (Variable): variable=internos
                  'desbaste_inicial'
                  bajada_broca := p[0,0,-0.012,0,0,0]
                  bajada := p[0,0,0.012,0,0,0]
                  MoveDirectionNode (selectedDirection=ZMinus toolParams=0.03, 0.035)
                    Until DISTANCE (allowActions=false deceleration=3 distanceNodeType=STOP) Distance=0.076; motionParameters(blendRadius=0)
                  Popup Message (haltProgram=false message=punto contacto alanzdo inputType=Text)
                  MoveDirectionNode (selectedDirection=ZPlus toolParams=0.003, 0.005)
                    Until DISTANCE (allowActions=false deceleration=3 distanceNodeType=STOP) Distance=0.002; motionParameters(blendRadius=0)
                  Wait Sleep waitTime=0.3
                  Set DigitalOutput pin=config_out[1]; digitalValue=1
                  Wait Sleep waitTime=0.3
                  Loop Counting (count=2) loopVariable(name=Loop_75)
                    bajar := pose_add(get_actual_tcp_pose(), bajada_broca)
                    Waypoint Waypoint (Variable): motionParameters(jointSpeed=1.047198 jointAcceleration=1.396263 cartesianSpeed=0.001 cartesianAcceleration=0.005); variable=bajar
                    subir := pose_sub(get_actual_tcp_pose(), bajada_broca)
                    Waypoint Waypoint (Variable): motionParameters(jointSpeed=1.047198 jointAcceleration=1.396263 cartesianSpeed=0.005 cartesianAcceleration=0.01); variable=subir
                    bajada_broca := pose_sub(bajada_broca, bajada)
                  MoveDirectionNode (selectedDirection=ZPlus toolParams=0.03, 0.035)
                    Until DISTANCE (allowActions=false deceleration=3 distanceNodeType=STOP) Distance=0.06; motionParameters(blendRadius=0)
                  Set DigitalOutput pin=config_out[1]; digitalValue=0
                  barreno_actual := barreno_actual+1
                  Call Quitar_broca
                  Call Poner_broca
          Folder CD
            'desbaste_inicial'
            bajada_broca := p[0,0,-0.012,0,0,0]
            barrenos_menos1 := 8
            barreno_actual := 0
            Loop While (checkContinuously=false) expression=barreno_actual≤barrenos_menos1
              Folder Perforacion
                MoveL speed 100 mm/s, acceleration 500 mm/s^2 (useActiveTCP=true) feature=Base
                  internos := interpolate_pose(Linea2_C, Linea2_D, barreno_actual/barrenos_menos1)
                  Waypoint Waypoint (Variable): variable=internos
                  'desbaste_inicial'
                  bajada_broca := p[0,0,-0.012,0,0,0]
                  bajada := p[0,0,0.012,0,0,0]
                  MoveDirectionNode (selectedDirection=ZMinus toolParams=0.03, 0.035)
                    Until DISTANCE (allowActions=false deceleration=3 distanceNodeType=STOP) Distance=0.076; motionParameters(blendRadius=0)
                  Popup Message (haltProgram=false message=punto contacto alanzdo inputType=Text)
                  MoveDirectionNode (selectedDirection=ZPlus toolParams=0.003, 0.005)
                    Until DISTANCE (allowActions=false deceleration=3 distanceNodeType=STOP) Distance=0.002; motionParameters(blendRadius=0)
                  Wait Sleep waitTime=0.3
                  Set DigitalOutput pin=config_out[1]; digitalValue=1
                  Wait Sleep waitTime=0.3
                  Loop Counting (count=2) loopVariable(name=Loop_78)
                    bajar := pose_add(get_actual_tcp_pose(), bajada_broca)
                    Waypoint Waypoint (Variable): motionParameters(jointSpeed=1.047198 jointAcceleration=1.396263 cartesianSpeed=0.001 cartesianAcceleration=0.005); variable=bajar
                    subir := pose_sub(get_actual_tcp_pose(), bajada_broca)
                    Waypoint Waypoint (Variable): motionParameters(jointSpeed=1.047198 jointAcceleration=1.396263 cartesianSpeed=0.005 cartesianAcceleration=0.01); variable=subir
                    bajada_broca := pose_sub(bajada_broca, bajada)
                  MoveDirectionNode (selectedDirection=ZPlus toolParams=0.03, 0.035)
                    Until DISTANCE (allowActions=false deceleration=3 distanceNodeType=STOP) Distance=0.06; motionParameters(blendRadius=0)
                  Set DigitalOutput pin=config_out[1]; digitalValue=0
                  barreno_actual := barreno_actual+1
                  Call Quitar_broca
                  Call Poner_broca
          Folder EF
            'desbaste_inicial'
            bajada_broca := p[0,0,-0.012,0,0,0]
            barrenos_menos1 := 8
            barreno_actual := 0
            Loop While (checkContinuously=false) expression=barreno_actual≤barrenos_menos1
              Folder Perforacion
                MoveL speed 100 mm/s, acceleration 500 mm/s^2 (useActiveTCP=true) feature=Base
                  internos := interpolate_pose(Linea2_E, Linea2_F, barreno_actual/barrenos_menos1)
                  Waypoint Waypoint (Variable): variable=internos
                  'desbaste_inicial'
                  bajada_broca := p[0,0,-0.012,0,0,0]
                  bajada := p[0,0,0.012,0,0,0]
                  MoveDirectionNode (selectedDirection=ZMinus toolParams=0.03, 0.035)
                    Until DISTANCE (allowActions=false deceleration=3 distanceNodeType=STOP) Distance=0.076; motionParameters(blendRadius=0)
                  Popup Message (haltProgram=false message=punto contacto alanzdo inputType=Text)
                  MoveDirectionNode (selectedDirection=ZPlus toolParams=0.003, 0.005)
                    Until DISTANCE (allowActions=false deceleration=3 distanceNodeType=STOP) Distance=0.002; motionParameters(blendRadius=0)
                  Wait Sleep waitTime=0.3
                  Set DigitalOutput pin=config_out[1]; digitalValue=1
                  Wait Sleep waitTime=0.3
                  Loop Counting (count=2) loopVariable(name=Loop_80)
                    bajar := pose_add(get_actual_tcp_pose(), bajada_broca)
                    Waypoint Waypoint (Variable): motionParameters(jointSpeed=1.047198 jointAcceleration=1.396263 cartesianSpeed=0.001 cartesianAcceleration=0.005); variable=bajar
                    subir := pose_sub(get_actual_tcp_pose(), bajada_broca)
                    Waypoint Waypoint (Variable): motionParameters(jointSpeed=1.047198 jointAcceleration=1.396263 cartesianSpeed=0.005 cartesianAcceleration=0.01); variable=subir
                    bajada_broca := pose_sub(bajada_broca, bajada)
                  MoveDirectionNode (selectedDirection=ZPlus toolParams=0.03, 0.035)
                    Until DISTANCE (allowActions=false deceleration=3 distanceNodeType=STOP) Distance=0.06; motionParameters(blendRadius=0)
                  Set DigitalOutput pin=config_out[1]; digitalValue=0
                  barreno_actual := barreno_actual+1
                  If barreno_actual>barrenos_menos1
                    cambiar_broca := True
                  Call Quitar_broca
                  Call Poner_broca
        Popup Message (haltProgram=false message=Linea2 con media Terminada! inputType=Text)
      Folder Broca_3
        Folder Linea1
          Folder Marcar_puntos
            MoveL speed 100 mm/s, acceleration 500 mm/s^2 (useActiveTCP=true) feature=Base
              Waypoint Home2: TCP in base x=-476.229 y=0 z=568.737 mm, rx=2.0263 ry=-2.3929 rz=-0.0208 rad; joints [-32.551, -116.469, 98.413, 17.843, -302.102, -0.163] deg; TCP offset x=0.411 y=-218.298 z=37.994 mm, rx=1.558 ry=-0.1255 rz=0.1212 rad
              Waypoint Linea1_A: TCP in base x=-480.065 y=-215.567 z=110.155 mm, rx=2.0263 ry=-2.3929 rz=-0.0208 rad; joints [7.208, -100.641, 136.552, -36.178, -262.472, -0.269] deg; TCP offset x=0.411 y=-218.298 z=37.994 mm, rx=1.558 ry=-0.1255 rz=0.1212 rad
              Waypoint Linea1_B: TCP in base x=-683.26 y=-215.006 z=110.473 mm, rx=2.0263 ry=-2.3929 rz=-0.0208 rad; joints [4.504, -82.11, 118.563, -36.711, -265.183, -0.242] deg
              Waypoint Linea1_C: TCP in base x=-708.66 y=-214.986 z=110.511 mm, rx=2.0264 ry=-2.3929 rz=-0.0208 rad; joints [4.302, -80.013, 116.028, -36.271, -265.387, -0.241] deg
              Waypoint Linea1_D: TCP in base x=-911.542 y=-214.533 z=110.306 mm, rx=2.0263 ry=-2.3929 rz=-0.0209 rad; joints [3.146, -63.772, 93.392, -29.877, -266.531, -0.235] deg
              Waypoint Linea1_E: TCP in base x=-936.518 y=-214.589 z=110.515 mm, rx=2.0263 ry=-2.3929 rz=-0.0209 rad; joints [3.051, -61.764, 90.233, -28.728, -266.622, -0.234] deg
              Waypoint Linea1_F: TCP in base x=-1139.514 y=-213.881 z=110.127 mm, rx=2.0263 ry=-2.3929 rz=-0.0209 rad; joints [2.389, -43.641, 59.472, -16.09, -267.256, -0.236] deg
          Folder AB
            'desbaste_inicial'
            bajada_broca := p[0,0,-0.012,0,0,0]
            barrenos_menos1 := 8
            barreno_actual := 0
            Loop While (checkContinuously=false) expression=barreno_actual≤barrenos_menos1
              Folder Perforacion
                MoveL speed 100 mm/s, acceleration 500 mm/s^2 (useActiveTCP=true) feature=Base
                  internos := interpolate_pose(Linea1_A, Linea1_B, barreno_actual/barrenos_menos1)
                  Waypoint Waypoint (Variable): variable=internos
                  'desbaste_inicial'
                  bajada_broca := p[0,0,-0.024,0,0,0]
                  bajada := p[0,0,0.024,0,0,0]
                  MoveDirectionNode (selectedDirection=ZMinus toolParams=0.03, 0.035)
                    Until DISTANCE (allowActions=false deceleration=3 distanceNodeType=STOP) Distance=0.072; motionParameters(blendRadius=0)
                  Popup Message (haltProgram=false message=punto contacto alanzdo inputType=Text)
                  MoveDirectionNode (selectedDirection=ZPlus toolParams=0.003, 0.005)
                    Until DISTANCE (allowActions=false deceleration=3 distanceNodeType=STOP) Distance=0.002; motionParameters(blendRadius=0)
                  Wait Sleep waitTime=0.3
                  Set DigitalOutput pin=config_out[1]; digitalValue=1
                  Wait Sleep waitTime=0.3
                  Loop Counting (count=1) loopVariable(name=Loop_82)
                    bajar := pose_add(get_actual_tcp_pose(), bajada_broca)
                    Waypoint Waypoint (Variable): motionParameters(jointSpeed=1.047198 jointAcceleration=1.396263 cartesianSpeed=0.001 cartesianAcceleration=0.005); variable=bajar
                    subir := pose_sub(get_actual_tcp_pose(), bajada_broca)
                    Waypoint Waypoint (Variable): motionParameters(jointSpeed=1.047198 jointAcceleration=1.396263 cartesianSpeed=0.005 cartesianAcceleration=0.01); variable=subir
                    bajada_broca := pose_sub(bajada_broca, bajada)
                  MoveDirectionNode (selectedDirection=ZPlus toolParams=0.03, 0.035)
                    Until DISTANCE (allowActions=false deceleration=3 distanceNodeType=STOP) Distance=0.06; motionParameters(blendRadius=0)
                  Set DigitalOutput pin=config_out[1]; digitalValue=0
                  barreno_actual := barreno_actual+1
                  Call Quitar_broca
                  Call Poner_broca
          Folder CD
            'desbaste_inicial'
            bajada_broca := p[0,0,-0.012,0,0,0]
            barrenos_menos1 := 8
            barreno_actual := 0
            Loop While (checkContinuously=false) expression=barreno_actual≤barrenos_menos1
              Folder Perforacion
                MoveL speed 100 mm/s, acceleration 500 mm/s^2 (useActiveTCP=true) feature=Base
                  internos := interpolate_pose(Linea1_C, Linea1_D, barreno_actual/barrenos_menos1)
                  Waypoint Waypoint (Variable): variable=internos
                  'desbaste_inicial'
                  bajada_broca := p[0,0,-0.024,0,0,0]
                  bajada := p[0,0,0.024,0,0,0]
                  MoveDirectionNode (selectedDirection=ZMinus toolParams=0.03, 0.035)
                    Until DISTANCE (allowActions=false deceleration=3 distanceNodeType=STOP) Distance=0.072; motionParameters(blendRadius=0)
                  Popup Message (haltProgram=false message=punto contacto alanzdo inputType=Text)
                  MoveDirectionNode (selectedDirection=ZPlus toolParams=0.003, 0.005)
                    Until DISTANCE (allowActions=false deceleration=3 distanceNodeType=STOP) Distance=0.002; motionParameters(blendRadius=0)
                  Wait Sleep waitTime=0.3
                  Set DigitalOutput pin=config_out[1]; digitalValue=1
                  Wait Sleep waitTime=0.3
                  Loop Counting (count=1) loopVariable(name=Loop_85)
                    bajar := pose_add(get_actual_tcp_pose(), bajada_broca)
                    Waypoint Waypoint (Variable): motionParameters(jointSpeed=1.047198 jointAcceleration=1.396263 cartesianSpeed=0.001 cartesianAcceleration=0.005); variable=bajar
                    subir := pose_sub(get_actual_tcp_pose(), bajada_broca)
                    Waypoint Waypoint (Variable): motionParameters(jointSpeed=1.047198 jointAcceleration=1.396263 cartesianSpeed=0.005 cartesianAcceleration=0.01); variable=subir
                    bajada_broca := pose_sub(bajada_broca, bajada)
                  MoveDirectionNode (selectedDirection=ZPlus toolParams=0.03, 0.035)
                    Until DISTANCE (allowActions=false deceleration=3 distanceNodeType=STOP) Distance=0.06; motionParameters(blendRadius=0)
                  Set DigitalOutput pin=config_out[1]; digitalValue=0
                  barreno_actual := barreno_actual+1
                  Call Quitar_broca
                  Call Poner_broca
          Folder EF
            'desbaste_inicial'
            bajada_broca := p[0,0,-0.012,0,0,0]
            barrenos_menos1 := 8
            barreno_actual := 0
            Loop While (checkContinuously=false) expression=barreno_actual≤barrenos_menos1
              Folder Perforacion
                MoveL speed 100 mm/s, acceleration 500 mm/s^2 (useActiveTCP=true) feature=Base
                  internos := interpolate_pose(Linea1_E, Linea1_F, barreno_actual/barrenos_menos1)
                  Waypoint Waypoint (Variable): variable=internos
                  'desbaste_inicial'
                  bajada_broca := p[0,0,-0.024,0,0,0]
                  bajada := p[0,0,0.024,0,0,0]
                  MoveDirectionNode (selectedDirection=ZMinus toolParams=0.03, 0.035)
                    Until DISTANCE (allowActions=false deceleration=3 distanceNodeType=STOP) Distance=0.072; motionParameters(blendRadius=0)
                  Popup Message (haltProgram=false message=punto contacto alanzdo inputType=Text)
                  MoveDirectionNode (selectedDirection=ZPlus toolParams=0.003, 0.005)
                    Until DISTANCE (allowActions=false deceleration=3 distanceNodeType=STOP) Distance=0.002; motionParameters(blendRadius=0)
                  Wait Sleep waitTime=0.3
                  Set DigitalOutput pin=config_out[1]; digitalValue=1
                  Wait Sleep waitTime=0.3
                  Loop Counting (count=1) loopVariable(name=Loop_87)
                    bajar := pose_add(get_actual_tcp_pose(), bajada_broca)
                    Waypoint Waypoint (Variable): motionParameters(jointSpeed=1.047198 jointAcceleration=1.396263 cartesianSpeed=0.001 cartesianAcceleration=0.005); variable=bajar
                    subir := pose_sub(get_actual_tcp_pose(), bajada_broca)
                    Waypoint Waypoint (Variable): motionParameters(jointSpeed=1.047198 jointAcceleration=1.396263 cartesianSpeed=0.005 cartesianAcceleration=0.01); variable=subir
                    bajada_broca := pose_sub(bajada_broca, bajada)
                  MoveDirectionNode (selectedDirection=ZPlus toolParams=0.03, 0.035)
                    Until DISTANCE (allowActions=false deceleration=3 distanceNodeType=STOP) Distance=0.06; motionParameters(blendRadius=0)
                  Set DigitalOutput pin=config_out[1]; digitalValue=0
                  barreno_actual := barreno_actual+1
                  Call Quitar_broca
                  Call Poner_broca
        Popup Message (haltProgram=false message=Linea1 con full Terminada! inputType=Text)
        Folder Linea2
          Folder Marcar_puntos
            MoveL speed 100 mm/s, acceleration 500 mm/s^2 (useActiveTCP=true) feature=Base
              Waypoint Home2: TCP in base x=-476.229 y=0 z=568.737 mm, rx=2.0263 ry=-2.3929 rz=-0.0208 rad; joints [-32.551, -116.469, 98.413, 17.843, -302.102, -0.163] deg; TCP offset x=0.411 y=-218.298 z=37.994 mm, rx=1.558 ry=-0.1255 rz=0.1212 rad
              SuppressedNode
                Folder var
                  barrenos_hechos := 0
                  eje7 := 2
                  cambiar_broca := False
                  iniciando_prog := False
              SuppressedNode
                iniciando_prog := False
              SuppressedNode
                Call Quitar_broca
              SuppressedNode
                Call Poner_broca
              Waypoint Linea2_A: TCP in base x=-478.57 y=191.006 z=110.523 mm, rx=2.0263 ry=-2.3928 rz=-0.0209 rad; joints [-57.982, -102.694, 138.014, -35.673, -327.66, 0.098] deg; TCP offset x=0.411 y=-218.298 z=37.994 mm, rx=1.558 ry=-0.1255 rz=0.1212 rad
              Waypoint Linea2_B: TCP in base x=-681.936 y=191.002 z=110.452 mm, rx=2.0263 ry=-2.3929 rz=-0.0209 rad; joints [-37.869, -83.103, 119.731, -36.904, -307.554, -0.038] deg
              Waypoint Linea2_C: TCP in base x=-707.214 y=190.995 z=110.603 mm, rx=2.0262 ry=-2.3929 rz=-0.0208 rad; joints [-36.266, -80.967, 117.182, -36.489, -305.951, -0.043] deg
              Waypoint Linea2_D: TCP in base x=-910.192 y=191.479 z=110.348 mm, rx=2.0262 ry=-2.3928 rz=-0.0209 rad; joints [-27.02, -64.45, 94.432, -30.243, -296.696, -0.089] deg
              Waypoint Linea2_E: TCP in base x=-935.62 y=191.519 z=110.454 mm, rx=2.0261 ry=-2.3928 rz=-0.021 rad; joints [-26.177, -62.39, 91.226, -29.103, -295.849, -0.094] deg
              Waypoint Linea2_F: TCP in base x=-1138.395 y=191.499 z=110.212 mm, rx=2.0262 ry=-2.3928 rz=-0.021 rad; joints [-20.933, -44.304, 60.66, -16.618, -290.578, -0.121] deg
          Folder AB
            'desbaste_inicial'
            bajada_broca := p[0,0,-0.012,0,0,0]
            barrenos_menos1 := 8
            barreno_actual := 1
            Loop While (checkContinuously=false) expression=barreno_actual≤barrenos_menos1
              Folder Perforacion
                MoveL speed 100 mm/s, acceleration 500 mm/s^2 (useActiveTCP=true) feature=Base
                  internos := interpolate_pose(Linea2_A, Linea2_B, barreno_actual/barrenos_menos1)
                  Waypoint Waypoint (Variable): variable=internos
                  'desbaste_inicial'
                  bajada_broca := p[0,0,-0.024,0,0,0]
                  bajada := p[0,0,0.024,0,0,0]
                  MoveDirectionNode (selectedDirection=ZMinus toolParams=0.03, 0.035)
                    Until DISTANCE (allowActions=false deceleration=3 distanceNodeType=STOP) Distance=0.076; motionParameters(blendRadius=0)
                  Popup Message (haltProgram=false message=punto contacto alanzdo inputType=Text)
                  MoveDirectionNode (selectedDirection=ZPlus toolParams=0.003, 0.005)
                    Until DISTANCE (allowActions=false deceleration=3 distanceNodeType=STOP) Distance=0.002; motionParameters(blendRadius=0)
                  Wait Sleep waitTime=0.3
                  Set DigitalOutput pin=config_out[1]; digitalValue=1
                  Wait Sleep waitTime=0.3
                  Loop Counting (count=1) loopVariable(name=Loop_90)
                    bajar := pose_add(get_actual_tcp_pose(), bajada_broca)
                    Waypoint Waypoint (Variable): motionParameters(jointSpeed=1.047198 jointAcceleration=1.396263 cartesianSpeed=0.001 cartesianAcceleration=0.005); variable=bajar
                    subir := pose_sub(get_actual_tcp_pose(), bajada_broca)
                    Waypoint Waypoint (Variable): motionParameters(jointSpeed=1.047198 jointAcceleration=1.396263 cartesianSpeed=0.005 cartesianAcceleration=0.01); variable=subir
                    bajada_broca := pose_sub(bajada_broca, bajada)
                  MoveDirectionNode (selectedDirection=ZPlus toolParams=0.03, 0.035)
                    Until DISTANCE (allowActions=false deceleration=3 distanceNodeType=STOP) Distance=0.06; motionParameters(blendRadius=0)
                  Set DigitalOutput pin=config_out[1]; digitalValue=0
                  barreno_actual := barreno_actual+1
                  Call Quitar_broca
                  Call Poner_broca
          Folder CD
            'desbaste_inicial'
            bajada_broca := p[0,0,-0.012,0,0,0]
            barrenos_menos1 := 8
            barreno_actual := 0
            Loop While (checkContinuously=false) expression=barreno_actual≤barrenos_menos1
              Folder Perforacion
                MoveL speed 100 mm/s, acceleration 500 mm/s^2 (useActiveTCP=true) feature=Base
                  internos := interpolate_pose(Linea2_C, Linea2_D, barreno_actual/barrenos_menos1)
                  Waypoint Waypoint (Variable): variable=internos
                  'desbaste_inicial'
                  bajada_broca := p[0,0,-0.024,0,0,0]
                  bajada := p[0,0,0.024,0,0,0]
                  MoveDirectionNode (selectedDirection=ZMinus toolParams=0.03, 0.035)
                    Until DISTANCE (allowActions=false deceleration=3 distanceNodeType=STOP) Distance=0.076; motionParameters(blendRadius=0)
                  Popup Message (haltProgram=false message=punto contacto alanzdo inputType=Text)
                  MoveDirectionNode (selectedDirection=ZPlus toolParams=0.003, 0.005)
                    Until DISTANCE (allowActions=false deceleration=3 distanceNodeType=STOP) Distance=0.002; motionParameters(blendRadius=0)
                  Wait Sleep waitTime=0.3
                  Set DigitalOutput pin=config_out[1]; digitalValue=1
                  Wait Sleep waitTime=0.3
                  Loop Counting (count=1) loopVariable(name=Loop_92)
                    bajar := pose_add(get_actual_tcp_pose(), bajada_broca)
                    Waypoint Waypoint (Variable): motionParameters(jointSpeed=1.047198 jointAcceleration=1.396263 cartesianSpeed=0.001 cartesianAcceleration=0.005); variable=bajar
                    subir := pose_sub(get_actual_tcp_pose(), bajada_broca)
                    Waypoint Waypoint (Variable): motionParameters(jointSpeed=1.047198 jointAcceleration=1.396263 cartesianSpeed=0.005 cartesianAcceleration=0.01); variable=subir
                    bajada_broca := pose_sub(bajada_broca, bajada)
                  MoveDirectionNode (selectedDirection=ZPlus toolParams=0.03, 0.035)
                    Until DISTANCE (allowActions=false deceleration=3 distanceNodeType=STOP) Distance=0.06; motionParameters(blendRadius=0)
                  Set DigitalOutput pin=config_out[1]; digitalValue=0
                  barreno_actual := barreno_actual+1
                  Call Quitar_broca
                  Call Poner_broca
          Folder EF
            'desbaste_inicial'
            bajada_broca := p[0,0,-0.012,0,0,0]
            barrenos_menos1 := 8
            barreno_actual := 0
            Loop While (checkContinuously=false) expression=barreno_actual≤barrenos_menos1
              Folder Perforacion
                MoveL speed 100 mm/s, acceleration 500 mm/s^2 (useActiveTCP=true) feature=Base
                  internos := interpolate_pose(Linea2_E, Linea2_F, barreno_actual/barrenos_menos1)
                  Waypoint Waypoint (Variable): variable=internos
                  'desbaste_inicial'
                  bajada_broca := p[0,0,-0.024,0,0,0]
                  bajada := p[0,0,0.024,0,0,0]
                  MoveDirectionNode (selectedDirection=ZMinus toolParams=0.03, 0.035)
                    Until DISTANCE (allowActions=false deceleration=3 distanceNodeType=STOP) Distance=0.076; motionParameters(blendRadius=0)
                  Popup Message (haltProgram=false message=punto contacto alanzdo inputType=Text)
                  MoveDirectionNode (selectedDirection=ZPlus toolParams=0.015, 0.015)
                    Until DISTANCE (allowActions=false deceleration=3 distanceNodeType=STOP) Distance=0.002; motionParameters(blendRadius=0)
                  Wait Sleep waitTime=0.3
                  Set DigitalOutput pin=config_out[1]; digitalValue=1
                  Wait Sleep waitTime=0.3
                  Loop Counting (count=1) loopVariable(name=Loop_94)
                    bajar := pose_add(get_actual_tcp_pose(), bajada_broca)
                    Waypoint Waypoint (Variable): motionParameters(jointSpeed=1.047198 jointAcceleration=1.396263 cartesianSpeed=0.001 cartesianAcceleration=0.005); variable=bajar
                    subir := pose_sub(get_actual_tcp_pose(), bajada_broca)
                    Waypoint Waypoint (Variable): motionParameters(jointSpeed=1.047198 jointAcceleration=1.396263 cartesianSpeed=0.005 cartesianAcceleration=0.01); variable=subir
                    bajada_broca := pose_sub(bajada_broca, bajada)
                  MoveDirectionNode (selectedDirection=ZPlus toolParams=0.03, 0.035)
                    Until DISTANCE (allowActions=false deceleration=3 distanceNodeType=STOP) Distance=0.06; motionParameters(blendRadius=0)
                  Set DigitalOutput pin=config_out[1]; digitalValue=0
                  barreno_actual := barreno_actual+1
                  If barreno_actual>barrenos_menos1
                    cambiar_broca := True
                  Call Quitar_broca
                  Call Poner_broca
        Popup Message (haltProgram=false message=Linea2 con full Terminada! inputType=Text)
    Folder 600
      SuppressedNode
        Folder Broca_1
          Folder Linea7
            Folder Marcar_puntos
              MoveL speed 100 mm/s, acceleration 500 mm/s^2 (useActiveTCP=true) feature=Base
                Waypoint Home2: TCP in base x=-476.229 y=0 z=568.737 mm, rx=2.0263 ry=-2.3929 rz=-0.0208 rad; joints [-32.551, -116.469, 98.413, 17.843, -302.102, -0.163] deg; TCP offset x=0.411 y=-218.298 z=37.994 mm, rx=1.558 ry=-0.1255 rz=0.1212 rad
                Waypoint Linea7_A: TCP in base x=-749.561 y=-351.839 z=110.843 mm, rx=3.1084 ry=-0.3759 rz=-0.0174 rad; joints [1.917, -65.95, 96.598, -30.808, -353.455, -0.309] deg
                Waypoint Linea7_B: TCP in base x=-795.37 y=-351.638 z=110.748 mm, rx=3.1084 ry=-0.3758 rz=-0.0174 rad; joints [1.792, -62.243, 90.906, -28.822, -353.578, -0.309] deg
            Folder AB
              'desbaste_inicial'
              bajada_broca := p[0,0,-0.008,0,0,0]
              barrenos_menos1 := 2
              barreno_actual := 0
              Loop While (checkContinuously=false) expression=barreno_actual≤barrenos_menos1
                Folder Perforacion
                  MoveL speed 100 mm/s, acceleration 500 mm/s^2 (useActiveTCP=true) feature=Base
                    internos := interpolate_pose(Linea7_A, Linea7_B, barreno_actual/barrenos_menos1)
                    Waypoint Waypoint (Variable): variable=internos
                    'desbaste_inicial'
                    bajada_broca := p[0,0,-0.024,0,0,0]
                    bajada := p[0,0,0.024,0,0,0]
                    MoveDirectionNode (selectedDirection=ZMinus toolParams=0.1, 0.15)
                      Until DISTANCE (allowActions=false deceleration=3 distanceNodeType=STOP) Distance=0.071; motionParameters(blendRadius=0)
                    MoveDirectionNode (selectedDirection=ZMinus toolParams=0.01, 0.01)
                      Until TOOL_CONTACT_DETECTION (allowActions=false retraction=0 decelerationAcceleration=0.01 decelerationAngularAcceleration=34.906585)
                    Popup Message (haltProgram=false message=punto contacto alanzdo inputType=Text)
                    MoveDirectionNode (selectedDirection=ZPlus toolParams=0.003, 0.005)
                      Until DISTANCE (allowActions=false deceleration=3 distanceNodeType=STOP) Distance=0.002; motionParameters(blendRadius=0)
                    Wait Sleep waitTime=0.3
                    Set DigitalOutput pin=config_out[1]; digitalValue=1
                    Wait Sleep waitTime=0.3
                    Loop Counting (count=1) loopVariable=Loop_56
                      bajar := pose_add(get_actual_tcp_pose(), bajada_broca)
                      Waypoint Waypoint (Variable): motionParameters(jointSpeed=1.047198 jointAcceleration=1.396263 cartesianSpeed=0.001 cartesianAcceleration=0.005); variable=bajar
                      subir := pose_sub(get_actual_tcp_pose(), bajada_broca)
                      Waypoint Waypoint (Variable): motionParameters(jointSpeed=1.047198 jointAcceleration=1.396263 cartesianSpeed=0.005 cartesianAcceleration=0.01); variable=subir
                      bajada_broca := pose_sub(bajada_broca, bajada)
                    MoveDirectionNode (selectedDirection=ZPlus toolParams=0.1, 0.15)
                      Until DISTANCE (allowActions=false deceleration=3 distanceNodeType=STOP) Distance=0.08; motionParameters(blendRadius=0)
                    Set DigitalOutput pin=config_out[1]; digitalValue=0
                    barreno_actual := barreno_actual+1
                    Call Quitar_broca
                    Call Poner_broca
          Popup Message (haltProgram=false message=Linea7 con chica Terminada! inputType=Text)
          Folder Linea8
            Folder Marcar_puntos
              MoveL speed 100 mm/s, acceleration 500 mm/s^2 (useActiveTCP=true) feature=Base
                Waypoint Linea8_A: TCP in base x=-897.665 y=-351.421 z=110.406 mm, rx=3.1084 ry=-0.3758 rz=-0.0174 rad; joints [1.574, -53.621, 76.868, -23.4, -353.783, -0.317] deg; TCP offset x=0.411 y=-218.298 z=37.994 mm, rx=1.558 ry=-0.1255 rz=0.1212 rad
                Waypoint Linea8_B: TCP in base x=-1021.743 y=-350.913 z=110.77 mm, rx=3.1084 ry=-0.3758 rz=-0.0173 rad; joints [1.351, -41.656, 55.75, -14.225, -353.984, -0.335] deg; TCP offset x=0.411 y=-218.298 z=37.994 mm, rx=1.558 ry=-0.1255 rz=0.1212 rad
            Folder AB
              'desbaste_inicial'
              bajada_broca := p[0,0,-0.008,0,0,0]
              barrenos_menos1 := 5
              barreno_actual := 0
              Loop While (checkContinuously=false) expression=barreno_actual≤barrenos_menos1
                Folder Perforacion
                  MoveL speed 100 mm/s, acceleration 500 mm/s^2 (useActiveTCP=true) feature=Base
                    internos := interpolate_pose(Linea8_A, Linea8_B, barreno_actual/barrenos_menos1)
                    Waypoint Waypoint (Variable): variable=internos
                    'desbaste_inicial'
                    bajada_broca := p[0,0,-0.008,0,0,0]
                    bajada := p[0,0,0.008,0,0,0]
                    MoveDirectionNode (selectedDirection=ZMinus toolParams=0.1, 0.15)
                      Until DISTANCE (allowActions=false deceleration=3 distanceNodeType=STOP) Distance=0.071; motionParameters(blendRadius=0)
                    MoveDirectionNode (selectedDirection=ZMinus toolParams=0.01, 0.01)
                      Until TOOL_CONTACT_DETECTION (allowActions=false retraction=0 decelerationAcceleration=0.01 decelerationAngularAcceleration=34.906585)
                    Popup Message (haltProgram=false message=punto contacto alanzdo inputType=Text)
                    MoveDirectionNode (selectedDirection=ZPlus toolParams=0.003, 0.005)
                      Until DISTANCE (allowActions=false deceleration=3 distanceNodeType=STOP) Distance=0.002; motionParameters(blendRadius=0)
                    Wait Sleep waitTime=0.3
                    Set DigitalOutput pin=config_out[1]; digitalValue=1
                    Wait Sleep waitTime=0.3
                    SuppressedNode
                      Loop Counting (count=3) loopVariable(name=Loop_68)
                        bajar := pose_add(get_actual_tcp_pose(), bajada_broca)
                        Waypoint Waypoint (Variable): motionParameters(jointSpeed=1.047198 jointAcceleration=1.396263 cartesianSpeed=0.001 cartesianAcceleration=0.005); variable=bajar
                        subir := pose_sub(get_actual_tcp_pose(), bajada_broca)
                        Waypoint Waypoint (Variable): motionParameters(jointSpeed=1.047198 jointAcceleration=1.396263 cartesianSpeed=0.005 cartesianAcceleration=0.01); variable=subir
                        bajada_broca := pose_sub(bajada_broca, bajada)
                    MoveDirectionNode (selectedDirection=ZPlus toolParams=0.1, 0.15)
                      Until DISTANCE (allowActions=false deceleration=3 distanceNodeType=STOP) Distance=0.08; motionParameters(blendRadius=0)
                    Set DigitalOutput pin=config_out[1]; digitalValue=0
                    barreno_actual := barreno_actual+1
                    SuppressedNode
                      Call Quitar_broca
                    SuppressedNode
                      Call Poner_broca
          Popup Message (haltProgram=false message=Linea8 con chica Terminada! inputType=Text)
          Folder Linea9
            Folder Marcar_puntos
              MoveL speed 100 mm/s, acceleration 500 mm/s^2 (useActiveTCP=true) feature=Base
                Waypoint Linea9_A: TCP in base x=-1101.64 y=-350.63 z=110.828 mm, rx=3.1084 ry=-0.3759 rz=-0.0174 rad; joints [1.234, -31.471, 36.669, -5.317, -354.073, -0.351] deg; TCP offset x=0.411 y=-218.298 z=37.994 mm, rx=1.558 ry=-0.1255 rz=0.1212 rad
                Waypoint Linea9_B: TCP in base x=-1151.202 y=-350.816 z=110.405 mm, rx=3.1084 ry=-0.3759 rz=-0.0174 rad; joints [1.184, -21.077, 16.327, 4.623, -354.093, -0.341] deg
            Folder AB
              'desbaste_inicial'
              bajada_broca := p[0,0,-0.008,0,0,0]
              barrenos_menos1 := 2
              barreno_actual := 0
              Loop While (checkContinuously=false) expression=barreno_actual≤barrenos_menos1
                Folder Perforacion
                  MoveL speed 100 mm/s, acceleration 500 mm/s^2 (useActiveTCP=true) feature=Base
                    internos := interpolate_pose(Linea9_A, Linea9_B, barreno_actual/barrenos_menos1)
                    Waypoint Waypoint (Variable): variable=internos
                    'desbaste_inicial'
                    bajada_broca := p[0,0,-0.008,0,0,0]
                    bajada := p[0,0,0.008,0,0,0]
                    MoveDirectionNode (selectedDirection=ZMinus toolParams=0.1, 0.15)
                      Until DISTANCE (allowActions=false deceleration=3 distanceNodeType=STOP) Distance=0.071; motionParameters(blendRadius=0)
                    MoveDirectionNode (selectedDirection=ZMinus toolParams=0.01, 0.01)
                      Until TOOL_CONTACT_DETECTION (allowActions=false retraction=0 decelerationAcceleration=0.01 decelerationAngularAcceleration=34.906585)
                    Popup Message (haltProgram=false message=punto contacto alanzdo inputType=Text)
                    MoveDirectionNode (selectedDirection=ZPlus toolParams=0.003, 0.005)
                      Until DISTANCE (allowActions=false deceleration=3 distanceNodeType=STOP) Distance=0.002; motionParameters(blendRadius=0)
                    Wait Sleep waitTime=0.3
                    Set DigitalOutput pin=config_out[1]; digitalValue=1
                    Wait Sleep waitTime=0.3
                    SuppressedNode
                      Loop Counting (count=3) loopVariable(name=Loop_74)
                        bajar := pose_add(get_actual_tcp_pose(), bajada_broca)
                        Waypoint Waypoint (Variable): motionParameters(jointSpeed=1.047198 jointAcceleration=1.396263 cartesianSpeed=0.001 cartesianAcceleration=0.005); variable=bajar
                        subir := pose_sub(get_actual_tcp_pose(), bajada_broca)
                        Waypoint Waypoint (Variable): motionParameters(jointSpeed=1.047198 jointAcceleration=1.396263 cartesianSpeed=0.005 cartesianAcceleration=0.01); variable=subir
                        bajada_broca := pose_sub(bajada_broca, bajada)
                    MoveDirectionNode (selectedDirection=ZPlus toolParams=0.1, 0.15)
                      Until DISTANCE (allowActions=false deceleration=3 distanceNodeType=STOP) Distance=0.08; motionParameters(blendRadius=0)
                    Set DigitalOutput pin=config_out[1]; digitalValue=0
                    barreno_actual := barreno_actual+1
                    SuppressedNode
                      Call Quitar_broca
                    SuppressedNode
                      Call Poner_broca
          Popup Message (haltProgram=false message=Linea9 con chica Terminada! inputType=Text)
          Folder Linea10
            Folder Marcar_puntos
              MoveL speed 100 mm/s, acceleration 500 mm/s^2 (useActiveTCP=true) feature=Base
                Waypoint Home2: TCP in base x=-476.229 y=0 z=568.737 mm, rx=2.0263 ry=-2.3929 rz=-0.0208 rad; joints [-32.551, -116.469, 98.413, 17.843, -302.102, -0.163] deg; TCP offset x=0.411 y=-218.298 z=37.994 mm, rx=1.558 ry=-0.1255 rz=0.1212 rad
                Waypoint Linea10_A: TCP in base x=-633.308 y=-317.691 z=110.995 mm, rx=3.1084 ry=-0.3759 rz=-0.0173 rad; joints [-0.882, -76.128, 110.969, -35.097, -356.258, -0.208] deg
                Waypoint Linea10_B: TCP in base x=-636.724 y=-266.696 z=110.314 mm, rx=2.0205 ry=-2.3939 rz=-0.0206 rad; joints [10.675, -83.921, 120.731, -37.208, -258.826, -0.176] deg
            Folder AB
              'desbaste_inicial'
              bajada_broca := p[0,0,-0.008,0,0,0]
              barrenos_menos1 := 2
              barreno_actual := 0
              Loop While (checkContinuously=false) expression=barreno_actual≤barrenos_menos1
                Folder Perforacion
                  MoveL speed 100 mm/s, acceleration 500 mm/s^2 (useActiveTCP=true) feature=Base
                    internos := interpolate_pose(Linea10_A, Linea10_B, barreno_actual/barrenos_menos1)
                    Waypoint Waypoint (Variable): variable=internos
                    'desbaste_inicial'
                    bajada_broca := p[0,0,-0.008,0,0,0]
                    bajada := p[0,0,0.008,0,0,0]
                    MoveDirectionNode (selectedDirection=ZMinus toolParams=0.1, 0.15)
                      Until DISTANCE (allowActions=false deceleration=3 distanceNodeType=STOP) Distance=0.071; motionParameters(blendRadius=0)
                    MoveDirectionNode (selectedDirection=ZMinus toolParams=0.001, 0.001)
                      Until TOOL_CONTACT_DETECTION (allowActions=false retraction=0 decelerationAcceleration=0.001 decelerationAngularAcceleration=34.906585)
                    Popup Message (haltProgram=false message=punto contacto alanzdo inputType=Text)
                    MoveDirectionNode (selectedDirection=ZPlus toolParams=0.003, 0.005)
                      Until DISTANCE (allowActions=false deceleration=3 distanceNodeType=STOP) Distance=0.002; motionParameters(blendRadius=0)
                    Wait Sleep waitTime=0.3
                    Set DigitalOutput pin=config_out[1]; digitalValue=1
                    Wait Sleep waitTime=0.3
                    SuppressedNode
                      Loop Counting (count=3) loopVariable(name=Loop_76)
                        bajar := pose_add(get_actual_tcp_pose(), bajada_broca)
                        Waypoint Waypoint (Variable): motionParameters(jointSpeed=1.047198 jointAcceleration=1.396263 cartesianSpeed=0.001 cartesianAcceleration=0.005); variable=bajar
                        subir := pose_sub(get_actual_tcp_pose(), bajada_broca)
                        Waypoint Waypoint (Variable): motionParameters(jointSpeed=1.047198 jointAcceleration=1.396263 cartesianSpeed=0.005 cartesianAcceleration=0.01); variable=subir
                        bajada_broca := pose_sub(bajada_broca, bajada)
                    MoveDirectionNode (selectedDirection=ZPlus toolParams=0.1, 0.15)
                      Until DISTANCE (allowActions=false deceleration=3 distanceNodeType=STOP) Distance=0.08; motionParameters(blendRadius=0)
                    Set DigitalOutput pin=config_out[1]; digitalValue=0
                    barreno_actual := barreno_actual+1
                    SuppressedNode
                      Call Quitar_broca
                    SuppressedNode
                      Call Poner_broca
          Popup Message (haltProgram=false message=Linea10 con chica Terminada! inputType=Text)
          Folder Linea11
            Folder Marcar_puntos
              MoveL speed 100 mm/s, acceleration 500 mm/s^2 (useActiveTCP=true) feature=Base
                Waypoint Linea11_A: TCP in base x=-636.133 y=-137.915 z=110.44 mm, rx=2.0204 ry=-2.394 rz=-0.0205 rad; joints [-4.201, -88.707, 125.915, -37.584, -273.698, -0.078] deg; TCP offset x=0.411 y=-218.298 z=37.994 mm, rx=1.558 ry=-0.1255 rz=0.1212 rad
                Waypoint Linea11_B: TCP in base x=-635.407 y=-82.609 z=110.403 mm, rx=2.0204 ry=-2.3939 rz=-0.0206 rad; joints [-11.006, -90.015, 127.249, -37.609, -280.504, -0.032] deg
            Folder AB
              'desbaste_inicial'
              bajada_broca := p[0,0,-0.008,0,0,0]
              barrenos_menos1 := 2
              barreno_actual := 0
              Loop While (checkContinuously=false) expression=barreno_actual≤barrenos_menos1
                Folder Perforacion
                  MoveL speed 100 mm/s, acceleration 500 mm/s^2 (useActiveTCP=true) feature=Base
                    SuppressedNode
                      If barreno_actual≟5
                        barreno_actual := barreno_actual+1
                    internos := interpolate_pose(Linea11_A, Linea11_B, barreno_actual/barrenos_menos1)
                    Waypoint Waypoint (Variable): variable=internos
                    'desbaste_inicial'
                    bajada_broca := p[0,0,-0.008,0,0,0]
                    bajada := p[0,0,0.008,0,0,0]
                    MoveDirectionNode (selectedDirection=ZMinus toolParams=0.1, 0.15)
                      Until DISTANCE (allowActions=false deceleration=3 distanceNodeType=STOP) Distance=0.071; motionParameters(blendRadius=0)
                    MoveDirectionNode (selectedDirection=ZMinus toolParams=0.001, 0.001)
                      Until TOOL_CONTACT_DETECTION (allowActions=false retraction=0 decelerationAcceleration=0.001 decelerationAngularAcceleration=34.906585)
                    Popup Message (haltProgram=false message=punto contacto alanzdo inputType=Text)
                    MoveDirectionNode (selectedDirection=ZPlus toolParams=0.003, 0.005)
                      Until DISTANCE (allowActions=false deceleration=3 distanceNodeType=STOP) Distance=0.002; motionParameters(blendRadius=0)
                    Wait Sleep waitTime=0.3
                    Set DigitalOutput pin=config_out[1]; digitalValue=1
                    Wait Sleep waitTime=0.3
                    SuppressedNode
                      Loop Counting (count=3) loopVariable=Loop_80
                        bajar := pose_add(get_actual_tcp_pose(), bajada_broca)
                        Waypoint Waypoint (Variable): motionParameters(jointSpeed=1.047198 jointAcceleration=1.396263 cartesianSpeed=0.001 cartesianAcceleration=0.005); variable=bajar
                        subir := pose_sub(get_actual_tcp_pose(), bajada_broca)
                        Waypoint Waypoint (Variable): motionParameters(jointSpeed=1.047198 jointAcceleration=1.396263 cartesianSpeed=0.005 cartesianAcceleration=0.01); variable=subir
                        bajada_broca := pose_sub(bajada_broca, bajada)
                    MoveDirectionNode (selectedDirection=ZPlus toolParams=0.1, 0.15)
                      Until DISTANCE (allowActions=false deceleration=3 distanceNodeType=STOP) Distance=0.08; motionParameters(blendRadius=0)
                    Set DigitalOutput pin=config_out[1]; digitalValue=0
                    barreno_actual := barreno_actual+1
                    SuppressedNode
                      Call Quitar_broca
                    SuppressedNode
                      Call Poner_broca
          Popup Message (haltProgram=false message=Linea11 con chica Terminada! inputType=Text)
          Folder Linea12
            Folder Marcar_puntos
              MoveL speed 100 mm/s, acceleration 500 mm/s^2 (useActiveTCP=true) feature=Base
                Waypoint Linea12_A: TCP in base x=-635.349 y=-59.56 z=110.675 mm, rx=2.0204 ry=-2.3939 rz=-0.0205 rad; joints [-13.849, -90.386, 127.583, -37.571, -283.348, -0.016] deg
                Waypoint Linea12_B: TCP in base x=-634.713 y=114.181 z=110.553 mm, rx=2.0204 ry=-2.3939 rz=-0.0206 rad; joints [-33.919, -89.532, 126.745, -37.627, -303.419, 0.135] deg
            Folder AB
              'desbaste_inicial'
              bajada_broca := p[0,0,-0.008,0,0,0]
              barrenos_menos1 := 7
              barreno_actual := 0
              Loop While (checkContinuously=false) expression=barreno_actual≤barrenos_menos1
                Folder Perforacion
                  MoveL speed 100 mm/s, acceleration 500 mm/s^2 (useActiveTCP=true) feature=Base
                    If barreno_actual≟2
                      barreno_actual := barreno_actual+1
                    internos := interpolate_pose(Linea12_A, Linea12_B, barreno_actual/barrenos_menos1)
                    Waypoint Waypoint (Variable): variable=internos
                    'desbaste_inicial'
                    bajada_broca := p[0,0,-0.008,0,0,0]
                    bajada := p[0,0,0.008,0,0,0]
                    MoveDirectionNode (selectedDirection=ZMinus toolParams=0.1, 0.15)
                      Until DISTANCE (allowActions=false deceleration=3 distanceNodeType=STOP) Distance=0.071; motionParameters(blendRadius=0)
                    MoveDirectionNode (selectedDirection=ZMinus toolParams=0.001, 0.001)
                      Until TOOL_CONTACT_DETECTION (allowActions=false retraction=0 decelerationAcceleration=0.001 decelerationAngularAcceleration=34.906585)
                    Popup Message (haltProgram=false message=punto contacto alanzdo inputType=Text)
                    MoveDirectionNode (selectedDirection=ZPlus toolParams=0.003, 0.005)
                      Until DISTANCE (allowActions=false deceleration=3 distanceNodeType=STOP) Distance=0.002; motionParameters(blendRadius=0)
                    Wait Sleep waitTime=0.3
                    Set DigitalOutput pin=config_out[1]; digitalValue=1
                    Wait Sleep waitTime=0.3
                    SuppressedNode
                      Loop Counting (count=3) loopVariable=Loop_78
                        bajar := pose_add(get_actual_tcp_pose(), bajada_broca)
                        Waypoint Waypoint (Variable): motionParameters(jointSpeed=1.047198 jointAcceleration=1.396263 cartesianSpeed=0.001 cartesianAcceleration=0.005); variable=bajar
                        subir := pose_sub(get_actual_tcp_pose(), bajada_broca)
                        Waypoint Waypoint (Variable): motionParameters(jointSpeed=1.047198 jointAcceleration=1.396263 cartesianSpeed=0.005 cartesianAcceleration=0.01); variable=subir
                        bajada_broca := pose_sub(bajada_broca, bajada)
                    MoveDirectionNode (selectedDirection=ZPlus toolParams=0.1, 0.15)
                      Until DISTANCE (allowActions=false deceleration=3 distanceNodeType=STOP) Distance=0.08; motionParameters(blendRadius=0)
                    Set DigitalOutput pin=config_out[1]; digitalValue=0
                    barreno_actual := barreno_actual+1
                    SuppressedNode
                      Call Quitar_broca
                    SuppressedNode
                      Call Poner_broca
          Popup Message (haltProgram=false message=Linea12 con chica Terminada! inputType=Text)
          Folder Linea13
            Folder Marcar_puntos
              MoveL speed 100 mm/s, acceleration 500 mm/s^2 (useActiveTCP=true) feature=Base
                Waypoint Linea13_A: TCP in base x=-634.623 y=269.838 z=110.202 mm, rx=2.0205 ry=-2.3939 rz=-0.0206 rad; joints [-47.693, -84.101, 120.951, -37.343, -317.193, 0.28] deg
                Waypoint Linea13_B: TCP in base x=-634.043 y=326.314 z=110.496 mm, rx=2.0205 ry=-2.3939 rz=-0.0206 rad; joints [-51.641, -81.48, 117.853, -36.903, -321.141, 0.338] deg
            Folder AB
              'desbaste_inicial'
              bajada_broca := p[0,0,-0.008,0,0,0]
              barrenos_menos1 := 2
              barreno_actual := 0
              Loop While (checkContinuously=false) expression=barreno_actual≤barrenos_menos1
                Folder Perforacion
                  MoveL speed 100 mm/s, acceleration 500 mm/s^2 (useActiveTCP=true) feature=Base
                    SuppressedNode
                      If barreno_actual≟2
                        barreno_actual := barreno_actual+1
                    internos := interpolate_pose(Linea13_A, Linea13_B, barreno_actual/barrenos_menos1)
                    Waypoint Waypoint (Variable): variable=internos
                    'desbaste_inicial'
                    bajada_broca := p[0,0,-0.008,0,0,0]
                    bajada := p[0,0,0.008,0,0,0]
                    MoveDirectionNode (selectedDirection=ZMinus toolParams=0.1, 0.15)
                      Until DISTANCE (allowActions=false deceleration=3 distanceNodeType=STOP) Distance=0.071; motionParameters(blendRadius=0)
                    MoveDirectionNode (selectedDirection=ZMinus toolParams=0.001, 0.001)
                      Until TOOL_CONTACT_DETECTION (allowActions=false retraction=0 decelerationAcceleration=0.001 decelerationAngularAcceleration=34.906585)
                    Popup Message (haltProgram=false message=punto contacto alanzdo inputType=Text)
                    MoveDirectionNode (selectedDirection=ZPlus toolParams=0.003, 0.005)
                      Until DISTANCE (allowActions=false deceleration=3 distanceNodeType=STOP) Distance=0.002; motionParameters(blendRadius=0)
                    Wait Sleep waitTime=0.3
                    Set DigitalOutput pin=config_out[1]; digitalValue=1
                    Wait Sleep waitTime=0.3
                    SuppressedNode
                      Loop Counting (count=3) loopVariable=Loop_82
                        bajar := pose_add(get_actual_tcp_pose(), bajada_broca)
                        Waypoint Waypoint (Variable): motionParameters(jointSpeed=1.047198 jointAcceleration=1.396263 cartesianSpeed=0.001 cartesianAcceleration=0.005); variable=bajar
                        subir := pose_sub(get_actual_tcp_pose(), bajada_broca)
                        Waypoint Waypoint (Variable): motionParameters(jointSpeed=1.047198 jointAcceleration=1.396263 cartesianSpeed=0.005 cartesianAcceleration=0.01); variable=subir
                        bajada_broca := pose_sub(bajada_broca, bajada)
                    MoveDirectionNode (selectedDirection=ZPlus toolParams=0.1, 0.15)
                      Until DISTANCE (allowActions=false deceleration=3 distanceNodeType=STOP) Distance=0.08; motionParameters(blendRadius=0)
                    Set DigitalOutput pin=config_out[1]; digitalValue=0
                    barreno_actual := barreno_actual+1
                    SuppressedNode
                      Call Quitar_broca
                    SuppressedNode
                      Call Poner_broca
          Popup Message (haltProgram=false message=Linea13 con chica Terminada! inputType=Text)
          Folder Linea14
            Folder Marcar_puntos
              MoveL speed 100 mm/s, acceleration 500 mm/s^2 (useActiveTCP=true) feature=Base
                Waypoint Linea14_A: TCP in base x=-633.963 y=349.887 z=111.384 mm, rx=2.0205 ry=-2.3938 rz=-0.0205 rad; joints [-53.122, -80.339, 116.362, -36.569, -322.623, 0.363] deg
                Waypoint Linea14_B: TCP in base x=-633.711 y=492.58 z=110.745 mm, rx=2.0205 ry=-2.3939 rz=-0.0205 rad; joints [-60.426, -72.306, 105.929, -34.278, -329.923, 0.504] deg; TCP offset x=0.411 y=-218.298 z=37.994 mm, rx=1.558 ry=-0.1255 rz=0.1212 rad
            Folder AB
              'desbaste_inicial'
              bajada_broca := p[0,0,-0.008,0,0,0]
              barrenos_menos1 := 5
              barreno_actual := 0
              Loop While (checkContinuously=false) expression=barreno_actual≤barrenos_menos1
                Folder Perforacion
                  MoveL speed 100 mm/s, acceleration 500 mm/s^2 (useActiveTCP=true) feature=Base
                    If barreno_actual≟3
                      barreno_actual := barreno_actual+1
                    internos := interpolate_pose(Linea14_A, Linea14_B, barreno_actual/barrenos_menos1)
                    Waypoint Waypoint (Variable): variable=internos
                    'desbaste_inicial'
                    bajada_broca := p[0,0,-0.008,0,0,0]
                    bajada := p[0,0,0.008,0,0,0]
                    MoveDirectionNode (selectedDirection=ZMinus toolParams=0.1, 0.15)
                      Until DISTANCE (allowActions=false deceleration=3 distanceNodeType=STOP) Distance=0.071; motionParameters(blendRadius=0)
                    MoveDirectionNode (selectedDirection=ZMinus toolParams=0.001, 0.001)
                      Until TOOL_CONTACT_DETECTION (allowActions=false retraction=0 decelerationAcceleration=0.001 decelerationAngularAcceleration=34.906585)
                    Popup Message (haltProgram=false message=punto contacto alanzdo inputType=Text)
                    MoveDirectionNode (selectedDirection=ZPlus toolParams=0.003, 0.005)
                      Until DISTANCE (allowActions=false deceleration=3 distanceNodeType=STOP) Distance=0.002; motionParameters(blendRadius=0)
                    Wait Sleep waitTime=0.3
                    Set DigitalOutput pin=config_out[1]; digitalValue=1
                    Wait Sleep waitTime=0.3
                    SuppressedNode
                      Loop Counting (count=3) loopVariable(name=Loop_84)
                        bajar := pose_add(get_actual_tcp_pose(), bajada_broca)
                        Waypoint Waypoint (Variable): motionParameters(jointSpeed=1.047198 jointAcceleration=1.396263 cartesianSpeed=0.001 cartesianAcceleration=0.005); variable=bajar
                        subir := pose_sub(get_actual_tcp_pose(), bajada_broca)
                        Waypoint Waypoint (Variable): motionParameters(jointSpeed=1.047198 jointAcceleration=1.396263 cartesianSpeed=0.005 cartesianAcceleration=0.01); variable=subir
                        bajada_broca := pose_sub(bajada_broca, bajada)
                    MoveDirectionNode (selectedDirection=ZPlus toolParams=0.1, 0.15)
                      Until DISTANCE (allowActions=false deceleration=3 distanceNodeType=STOP) Distance=0.08; motionParameters(blendRadius=0)
                    Set DigitalOutput pin=config_out[1]; digitalValue=0
                    barreno_actual := barreno_actual+1
                    SuppressedNode
                      Call Quitar_broca
                    SuppressedNode
                      Call Poner_broca
          Popup Message (haltProgram=false message=Linea14 con chica Terminada! inputType=Text)
          Folder Linea15
            Folder Marcar_puntos
              MoveL speed 100 mm/s, acceleration 500 mm/s^2 (useActiveTCP=true) feature=Base
                Waypoint Linea15_A: TCP in base x=-633.318 y=515.44 z=110.158 mm, rx=2.0204 ry=-2.394 rz=-0.0205 rad; joints [-61.401, -70.918, 104.049, -33.805, -330.892, 0.526] deg
                Waypoint Linea15_B: TCP in base x=-632.971 y=593.971 z=110.611 mm, rx=2.0204 ry=-2.3939 rz=-0.0206 rad; joints [-64.313, -66.034, 96.849, -31.559, -333.804, 0.606] deg
            Folder AB
              'desbaste_inicial'
              bajada_broca := p[0,0,-0.008,0,0,0]
              barrenos_menos1 := 3
              barreno_actual := 0
              Loop While (checkContinuously=false) expression=barreno_actual≤barrenos_menos1
                Folder Perforacion
                  MoveL speed 100 mm/s, acceleration 500 mm/s^2 (useActiveTCP=true) feature=Base
                    SuppressedNode
                      If barreno_actual≟3
                        barreno_actual := barreno_actual+1
                    internos := interpolate_pose(Linea15_A, Linea15_B, barreno_actual/barrenos_menos1)
                    Waypoint Waypoint (Variable): variable=internos
                    'desbaste_inicial'
                    bajada_broca := p[0,0,-0.008,0,0,0]
                    bajada := p[0,0,0.008,0,0,0]
                    MoveDirectionNode (selectedDirection=ZMinus toolParams=0.1, 0.15)
                      Until DISTANCE (allowActions=false deceleration=3 distanceNodeType=STOP) Distance=0.071; motionParameters(blendRadius=0)
                    MoveDirectionNode (selectedDirection=ZMinus toolParams=0.001, 0.001)
                      Until TOOL_CONTACT_DETECTION (allowActions=false retraction=0 decelerationAcceleration=0.001 decelerationAngularAcceleration=34.906585)
                    Popup Message (haltProgram=false message=punto contacto alanzdo inputType=Text)
                    MoveDirectionNode (selectedDirection=ZPlus toolParams=0.003, 0.005)
                      Until DISTANCE (allowActions=false deceleration=3 distanceNodeType=STOP) Distance=0.002; motionParameters(blendRadius=0)
                    Wait Sleep waitTime=0.3
                    Set DigitalOutput pin=config_out[1]; digitalValue=1
                    Wait Sleep waitTime=0.3
                    SuppressedNode
                      Loop Counting (count=3) loopVariable(name=Loop_86)
                        bajar := pose_add(get_actual_tcp_pose(), bajada_broca)
                        Waypoint Waypoint (Variable): motionParameters(jointSpeed=1.047198 jointAcceleration=1.396263 cartesianSpeed=0.001 cartesianAcceleration=0.005); variable=bajar
                        subir := pose_sub(get_actual_tcp_pose(), bajada_broca)
                        Waypoint Waypoint (Variable): motionParameters(jointSpeed=1.047198 jointAcceleration=1.396263 cartesianSpeed=0.005 cartesianAcceleration=0.01); variable=subir
                        bajada_broca := pose_sub(bajada_broca, bajada)
                    MoveDirectionNode (selectedDirection=ZPlus toolParams=0.1, 0.15)
                      Until DISTANCE (allowActions=false deceleration=3 distanceNodeType=STOP) Distance=0.08; motionParameters(blendRadius=0)
                    Set DigitalOutput pin=config_out[1]; digitalValue=0
                    barreno_actual := barreno_actual+1
                    SuppressedNode
                      Call Quitar_broca
                    SuppressedNode
                      Call Poner_broca
          Popup Message (haltProgram=false message=Linea15 con chica Terminada! inputType=Text)
          Folder Linea16
            Folder Marcar_puntos
              MoveL speed 100 mm/s, acceleration 500 mm/s^2 (useActiveTCP=true) feature=Base
                Waypoint Linea16_A: TCP in base x=-469.659 y=618.24 z=110.223 mm, rx=-0.2145 ry=-3.1278 rz=-0.004 rad; joints [-60.494, -74.578, 108.875, -33.964, -241.822, 0.658] deg
                Waypoint Linea16_B: TCP in base x=-493.719 y=618.586 z=110.183 mm, rx=-0.2145 ry=-3.1278 rz=-0.004 rad; joints [-58.661, -73.102, 106.872, -33.43, -239.985, 0.672] deg
            Folder AB
              'desbaste_inicial'
              bajada_broca := p[0,0,-0.008,0,0,0]
              barrenos_menos1 := 1
              barreno_actual := 0
              Loop While (checkContinuously=false) expression=barreno_actual≤barrenos_menos1
                Folder Perforacion
                  MoveL speed 100 mm/s, acceleration 500 mm/s^2 (useActiveTCP=true) feature=Base
                    SuppressedNode
                      If barreno_actual≟3
                        barreno_actual := barreno_actual+1
                    internos := interpolate_pose(Linea16_A, Linea16_B, barreno_actual/barrenos_menos1)
                    Waypoint Waypoint (Variable): variable=internos
                    'desbaste_inicial'
                    bajada_broca := p[0,0,-0.008,0,0,0]
                    bajada := p[0,0,0.008,0,0,0]
                    MoveDirectionNode (selectedDirection=ZMinus toolParams=0.1, 0.15)
                      Until DISTANCE (allowActions=false deceleration=3 distanceNodeType=STOP) Distance=0.071; motionParameters(blendRadius=0)
                    MoveDirectionNode (selectedDirection=ZMinus toolParams=0.001, 0.001)
                      Until TOOL_CONTACT_DETECTION (allowActions=false retraction=0 decelerationAcceleration=0.001 decelerationAngularAcceleration=34.906585)
                    Popup Message (haltProgram=false message=punto contacto alanzdo inputType=Text)
                    MoveDirectionNode (selectedDirection=ZPlus toolParams=0.003, 0.005)
                      Until DISTANCE (allowActions=false deceleration=3 distanceNodeType=STOP) Distance=0.002; motionParameters(blendRadius=0)
                    Wait Sleep waitTime=0.3
                    Set DigitalOutput pin=config_out[1]; digitalValue=1
                    Wait Sleep waitTime=0.3
                    SuppressedNode
                      Loop Counting (count=3) loopVariable(name=Loop_88)
                        bajar := pose_add(get_actual_tcp_pose(), bajada_broca)
                        Waypoint Waypoint (Variable): motionParameters(jointSpeed=1.047198 jointAcceleration=1.396263 cartesianSpeed=0.001 cartesianAcceleration=0.005); variable=bajar
                        subir := pose_sub(get_actual_tcp_pose(), bajada_broca)
                        Waypoint Waypoint (Variable): motionParameters(jointSpeed=1.047198 jointAcceleration=1.396263 cartesianSpeed=0.005 cartesianAcceleration=0.01); variable=subir
                        bajada_broca := pose_sub(bajada_broca, bajada)
                    MoveDirectionNode (selectedDirection=ZPlus toolParams=0.1, 0.15)
                      Until DISTANCE (allowActions=false deceleration=3 distanceNodeType=STOP) Distance=0.08; motionParameters(blendRadius=0)
                    Set DigitalOutput pin=config_out[1]; digitalValue=0
                    barreno_actual := barreno_actual+1
                    SuppressedNode
                      Call Quitar_broca
                    SuppressedNode
                      Call Poner_broca
          Popup Message (haltProgram=false message=Linea16 con chica Terminada! inputType=Text)
          Folder Linea17
            Folder Marcar_puntos
              MoveL speed 100 mm/s, acceleration 500 mm/s^2 (useActiveTCP=true) feature=Base
                Waypoint Linea17_A: TCP in base x=-523.229 y=618.283 z=110.575 mm, rx=-0.2145 ry=-3.1278 rz=-0.0039 rad; joints [-56.495, -71.324, 104.348, -32.678, -237.82, 0.686] deg
                Waypoint Linea17_B: TCP in base x=-574.505 y=618.78 z=110.128 mm, rx=-0.2145 ry=-3.1278 rz=-0.0039 rad; joints [-53.062, -68.029, 99.656, -31.269, -234.384, 0.712] deg
            Folder AB
              'desbaste_inicial'
              bajada_broca := p[0,0,-0.008,0,0,0]
              barrenos_menos1 := 2
              barreno_actual := 0
              Loop While (checkContinuously=false) expression=barreno_actual≤barrenos_menos1
                Folder Perforacion
                  MoveL speed 100 mm/s, acceleration 500 mm/s^2 (useActiveTCP=true) feature=Base
                    SuppressedNode
                      If barreno_actual≟3
                        barreno_actual := barreno_actual+1
                    internos := interpolate_pose(Linea17_A, Linea17_B, barreno_actual/barrenos_menos1)
                    Waypoint Waypoint (Variable): variable=internos
                    'desbaste_inicial'
                    bajada_broca := p[0,0,-0.008,0,0,0]
                    bajada := p[0,0,0.008,0,0,0]
                    MoveDirectionNode (selectedDirection=ZMinus toolParams=0.1, 0.15)
                      Until DISTANCE (allowActions=false deceleration=3 distanceNodeType=STOP) Distance=0.071; motionParameters(blendRadius=0)
                    MoveDirectionNode (selectedDirection=ZMinus toolParams=0.001, 0.001)
                      Until TOOL_CONTACT_DETECTION (allowActions=false retraction=0 decelerationAcceleration=0.001 decelerationAngularAcceleration=34.906585)
                    Popup Message (haltProgram=false message=punto contacto alanzdo inputType=Text)
                    MoveDirectionNode (selectedDirection=ZPlus toolParams=0.1, 0.15)
                      Until DISTANCE (allowActions=false deceleration=3 distanceNodeType=STOP) Distance=0.002; motionParameters(blendRadius=0)
                    Wait Sleep waitTime=0.3
                    Set DigitalOutput pin=config_out[1]; digitalValue=1
                    Wait Sleep waitTime=0.3
                    SuppressedNode
                      Loop Counting (count=3) loopVariable=Loop_90
                        bajar := pose_add(get_actual_tcp_pose(), bajada_broca)
                        Waypoint Waypoint (Variable): motionParameters(jointSpeed=1.047198 jointAcceleration=1.396263 cartesianSpeed=0.001 cartesianAcceleration=0.005); variable=bajar
                        subir := pose_sub(get_actual_tcp_pose(), bajada_broca)
                        Waypoint Waypoint (Variable): motionParameters(jointSpeed=1.047198 jointAcceleration=1.396263 cartesianSpeed=0.005 cartesianAcceleration=0.01); variable=subir
                        bajada_broca := pose_sub(bajada_broca, bajada)
                    MoveDirectionNode (selectedDirection=ZPlus toolParams=0.03, 0.035)
                      Until DISTANCE (allowActions=false deceleration=3 distanceNodeType=STOP) Distance=0.08; motionParameters(blendRadius=0)
                    Set DigitalOutput pin=config_out[1]; digitalValue=0
                    barreno_actual := barreno_actual+1
                    SuppressedNode
                      Call Quitar_broca
